(* IEC 61131-3 sources: Industry-PLC-LLM/data/PLCBEAD_repo/PLCBEAD_PLCEmbed-main/PLC-BEAD/Source/OpenPLCv2 (part 3) *)

(* ---- CEXP.ST ---- *)
TYPE oscat_complex :
  STRUCT
	re : REAL;
	im : REAL;
  END_STRUCT;
END_TYPE

FUNCTION_BLOCK CEXP_Block
	VAR_INPUT
		X :	oscat_complex;
	END_VAR

	VAR_OUTPUT
		CEXP :	oscat_complex;
	END_VAR

	VAR
		Temp :	REAL;
	END_VAR

	temp := EXP(X.re);
	CEXP.re := temp * COS(X.im);
	CEXP.im := temp * SIN(X.im);

END_FUNCTION_BLOCK

PROGRAM program0
  VAR
    LocalVar0 : oscat_complex;
	LocalOUT  : oscat_complex;
	func_block : CEXP_Block;
  END_VAR
	func_block.X  := LocalVar0;
	func_block();
	LocalOUT := func_block.CEXP;
END_PROGRAM

CONFIGURATION Config0
  RESOURCE Res0 ON PLC
    TASK task0(INTERVAL := T#20ms,PRIORITY := 0);
    PROGRAM instance0 WITH task0 : program0;
  END_RESOURCE
END_CONFIGURATION

(* ---- CHARNAME.ST ---- *)
TYPE
  oscat_CHARNAMES	: ARRAY [1..11] OF STRING;
END_TYPE

FUNCTION_BLOCK SETUP_CHARNAMES_Block

	VAR_IN_OUT
		CHARNAMES :	oscat_CHARNAMES;
	END_VAR

	VAR
		init :	BOOL;
	END_VAR

	IF init THEN RETURN; END_IF;

	init := TRUE;

	CHARNAMES[01] := '123';
	CHARNAMES[02] := '456';
	CHARNAMES[03] := 'zgsdafasf';
	CHARNAMES[04] := 'sadfsdfa';
	CHARNAMES[05] := 'asdfdsafdfds';
	CHARNAMES[06] := 'sadfsdfsdf';
	CHARNAMES[07] := 'sfsfdfdddd';
	CHARNAMES[08] := 'dddddted';
	CHARNAMES[10] := 'wer';
	CHARNAMES[11] := 'werwer';

END_FUNCTION_BLOCK

FUNCTION_BLOCK CHR_TO_STRING_Block
	VAR_INPUT
		C :	BYTE;
	END_VAR

	VAR_OUTPUT
		CHR_TO_STRING :	STRING;
	END_VAR

	CHR_TO_STRING := BYTE_TO_STRING(C);

END_FUNCTION_BLOCK

FUNCTION_BLOCK CHARNAME_Block

	VAR_INPUT
		C :	BYTE;
	END_VAR

	VAR_OUTPUT
		CHARNAME :	STRING;
	END_VAR

	VAR
		CHARNAME2 :	STRING;
		pos :	INT;
		i :	INT;
		CHR_TO_STRING :	CHR_TO_STRING_Block;
		SETUP_CHARNAMES :	SETUP_CHARNAMES_Block;
		CHARNAMES :	oscat_CHARNAMES;
	END_VAR

	SETUP_CHARNAMES(CHARNAMES:=CHARNAMES);
	CHARNAMES:=SETUP_CHARNAMES.CHARNAMES;

	IF C <> BYTE#0 THEN
		(* construct search string from code followed by $ sign, also clear charname string*)
		CHR_TO_STRING(C:=C);
		CHARNAME := CHR_TO_STRING.CHR_TO_STRING;
		CHARNAME2 := CONCAT(CHARNAME,'&');
		CHARNAME := CONCAT(';', CHARNAME2);
		WHILE pos = 0 AND (i < 11) DO
			i := i + 1;
			pos := FIND(CHARNAMES[i], CHARNAME);
		END_WHILE;
		IF pos > 0 THEN
			CHARNAME := MID(CHARNAMES[i], 10, pos + 3);
			(* search for end of name and truncate *)
			pos := FIND(CHARNAME, ';');
			CHARNAME := LEFT(CHARNAME,pos - 1);
		ELSE
			CHR_TO_STRING(C:=C);
			CHARNAME := CHR_TO_STRING.CHR_TO_STRING;
		END_IF;
	ELSE
		CHARNAME := '';
	END_IF;

END_FUNCTION_BLOCK

PROGRAM program0
  VAR
	C :	BYTE;
	CHARNAME :	STRING;
	func_block : CHARNAME_Block;
  END_VAR
	func_block.C  :=C ;
	func_block();
	CHARNAME := func_block.CHARNAME;
END_PROGRAM

CONFIGURATION Config0
	RESOURCE Res0 ON PLC
		TASK task0(INTERVAL := T#20ms,PRIORITY := 0);
		PROGRAM instance0 WITH task0 : program0;
	END_RESOURCE
END_CONFIGURATION

(* ---- CHR_TO_STRING.ST ---- *)
FUNCTION_BLOCK CHR_TO_STRING_Block
	VAR_INPUT
		C :	BYTE;
	END_VAR

	VAR_OUTPUT
		CHR_TO_STRING :	STRING;
	END_VAR

	CHR_TO_STRING := BYTE_TO_STRING(C);

END_FUNCTION_BLOCK

PROGRAM program0
  VAR
    LocalVar0 : BYTE;
	LocalOUT  : STRING;
	func_block : CHR_TO_STRING_Block;
  END_VAR
	func_block.C  := LocalVar0;
	func_block();
	LocalOUT := func_block.CHR_TO_STRING;
END_PROGRAM

CONFIGURATION Config0
  RESOURCE Res0 ON PLC
    TASK task0(INTERVAL := T#20ms,PRIORITY := 0);
    PROGRAM instance0 WITH task0 : program0;
  END_RESOURCE
END_CONFIGURATION

(* ---- CINV.ST ---- *)
TYPE oscat_complex :
  STRUCT
	re : REAL;
	im : REAL;
  END_STRUCT;
END_TYPE

FUNCTION_BLOCK CINV_Block

	VAR_INPUT
		X :	oscat_complex;
	END_VAR

	VAR_OUTPUT
		CINV :	oscat_complex;
	END_VAR

	VAR
		temp :	REAL;
	END_VAR

	temp := X.re * X.re + X.im * X.im;
	IF temp = 0.0 THEN CINV.re := 0.0;CINV.im := 0.0;RETURN;END_IF;
	CINV.re := X.re / temp;
	CINV.im := -X.im / temp;

END_FUNCTION_BLOCK

PROGRAM program0
  VAR
    LocalVar0 : oscat_complex;
	LocalOUT  : oscat_complex;
	func_block : CINV_Block;
  END_VAR
	func_block.X  := LocalVar0;
	func_block();
	LocalOUT := func_block.CINV;
END_PROGRAM

CONFIGURATION Config0
  RESOURCE Res0 ON PLC
    TASK task0(INTERVAL := T#20ms,PRIORITY := 0);
    PROGRAM instance0 WITH task0 : program0;
  END_RESOURCE
END_CONFIGURATION

(* ---- CLEAN.ST ---- *)
FUNCTION_BLOCK CLEAN_Block
	VAR_INPUT
		IN :	STRING;
		CX :	STRING;
	END_VAR

	VAR_OUTPUT
		CLEAN :	STRING;
	END_VAR

	VAR
		pos :	INT;
		stop :	INT;
		char :	STRING;
	END_VAR

	CLEAN := IN;
	stop := LEN(in);
	pos := 1;
	WHILE pos <= stop DO
		char := MID(CLEAN, 1, pos);
		IF FIND(cx,char) > 0 THEN
			pos := pos + 1;
		ELSE
			CLEAN := DELETE(CLEAN, 1, pos);
			stop := stop - 1;
		END_IF;
	END_WHILE;

END_FUNCTION_BLOCK

PROGRAM program0
  VAR
    LocalVar0 : STRING;
    LocalVar1 : STRING;
	LocalOUT  : STRING;
	func_block : CLEAN_Block;
  END_VAR
	func_block.IN  := LocalVar0;
	func_block.CX := LocalVar1;
	func_block();
	LocalOUT := func_block.CLEAN;

END_PROGRAM

CONFIGURATION Config0
  RESOURCE Res0 ON PLC
    TASK task0(INTERVAL := T#20ms,PRIORITY := 0);
    PROGRAM instance0 WITH task0 : program0;
  END_RESOURCE
END_CONFIGURATION

(* ---- CLICK.ST ---- *)
FUNCTION_BLOCK SW_RECONFIG_Block

	VAR_INPUT
		IN :	BOOL;
		TD :	TIME;
		TR :	TIME;
	END_VAR

	VAR_OUTPUT
		Q :	BOOL;
	END_VAR

	VAR
		T1 :	TON;
		T2 :	TON;
		INV :	BOOL;
	END_VAR

	t1(in := IN, PT := TD);

	IF tr > t#0s THEN
		Q := t1.Q XOR inv;
		T2(in := Q, pt := TR);
		IF T2.Q THEN INV := NOT INV; END_IF;
	ELSE
		Q := t1.Q;
	END_IF;

END_FUNCTION_BLOCK

FUNCTION UDINT_TO_TIME2:TIME

	VAR_INPUT
		IN :	UDINT;
	END_VAR

	UDINT_TO_TIME2 := DINT_TO_TIME(UDINT_TO_DINT(IN));

END_FUNCTION

FUNCTION_BLOCK T_PLC_MS_block
	VAR_OUTPUT
		T_PLC_MS :	UDINT;
	END_VAR

	VAR_EXTERNAL
		PLC_TICKS_PER_SEC :	INT;
		PLC_SYS_TICK_CNT :	DINT;
	END_VAR

	VAR
		debug :	BOOL;(*Debug-Mode ON / OFF*)
		N :	INT;(*Debug-Faktor*)
		Offset :	UDINT;(*Debug-Offset*)
		temp :	DWORD := DWORD#1;(*Debug-Offset*)
		mode :	BOOL;(*modus*)
		faktor :	UDINT;(*Systemtakt-Faktor*)
		init :	BOOL;
		v_plc_ticks_per_sec :	UDINT;
		base :	UDINT := UDINT#1000;
	END_VAR

	IF init = FALSE THEN
		v_plc_ticks_per_sec := INT_TO_UDINT(PLC_TICKS_PER_SEC);
		IF v_plc_ticks_per_sec = UDINT#1024 THEN
			faktor := UDINT#1;
			mode := FALSE;
		ELSIF v_plc_ticks_per_sec > UDINT#0 THEN
			IF v_plc_ticks_per_sec <= base THEN
				faktor := base / v_plc_ticks_per_sec;
				mode := FALSE;
			ELSE
				faktor := v_plc_ticks_per_sec / base;
				mode := TRUE;
			END_IF;
		ELSE
			faktor := UDINT#1;
		END_IF;
		init := TRUE;
	END_IF;

	IF mode THEN
		T_PLC_MS := DINT_TO_UDINT(PLC_SYS_TICK_CNT) / faktor;
	ELSE
		T_PLC_MS := DINT_TO_UDINT(PLC_SYS_TICK_CNT) * faktor;
	END_IF;

	IF debug THEN
		T_PLC_MS := (DWORD_TO_UDINT(SHL(UDINT_TO_DWORD(T_PLC_MS),N) OR SHL(temp,N)) - UDINT#1) + Offset;
	END_IF;

END_FUNCTION_BLOCK

FUNCTION_BLOCK CLICK_Block

	VAR_INPUT
		IN :	BOOL;
		T_DEBOUNCE :	TIME := T#10ms;
		T_SHORT :	TIME := T#200ms;
		T_PAUSE :	TIME := T#500ms;
		T_RECONFIG :	TIME := T#1m;
	END_VAR

	VAR_OUTPUT
		Q :	BOOL;
		SINGLE :	BOOL;
		DOUBLE :	BOOL;
		TRIPLE :	BOOL;
		STATUS :	BYTE;
	END_VAR

	VAR
		s_in :	SW_RECONFIG_Block;
		tx :	TIME;
		state :	INT;
		last :	TIME;
		T_PLC_MS :	T_PLC_MS_Block;
	END_VAR

	s_in(in := in, TD := T_debounce, TR := T_reconfig);

	T_PLC_MS();
	tx:= UDINT_TO_TIME(T_PLC_MS.T_PLC_MS);

	IF s_in.Q XOR Q THEN
		last := tx;
		IF s_in.Q THEN state := state + 1; END_IF;
	END_IF;
	Q := s_in.Q;

	IF state > 0 THEN
		IF (Q AND tx - last > t_short) OR (NOT Q AND tx - last > t_pause) THEN
			CASE state OF
				1:	single := TRUE;
					status := BYTE#111;
				2:	double := TRUE;
					status := BYTE#112;
				3:	triple := TRUE;
					status := BYTE#113;
			END_CASE;
			state := 0;
		END_IF;
	ELSIF NOT q THEN
		single := FALSE;
		double := FALSE;
		triple := FALSE;
		status := BYTE#110;
		last := tx;
		state := 0;
	END_IF;

END_FUNCTION_BLOCK

PROGRAM program0
	VAR
		IN :	BOOL;
		T_DEBOUNCE :	TIME := T#10ms;
		T_SHORT :	TIME := T#200ms;
		T_PAUSE :	TIME := T#500ms;
		T_RECONFIG :	TIME := T#1m;
		Q :	BOOL;
		SINGLE :	BOOL;
		DOUBLE :	BOOL;
		TRIPLE :	BOOL;
		STATUS :	BYTE;

		func_block : CLICK_Block;
	END_VAR
	func_block.IN := IN;
	func_block.T_DEBOUNCE := T_DEBOUNCE;
	func_block.T_SHORT := T_SHORT;
	func_block.T_PAUSE := T_PAUSE;
	func_block.T_RECONFIG := T_RECONFIG;

	func_block();
	Q  := func_block.Q;
	SINGLE  := func_block.SINGLE;
	DOUBLE  := func_block.DOUBLE;
	TRIPLE  := func_block.TRIPLE;
	STATUS  := func_block.STATUS;
END_PROGRAM

CONFIGURATION Config0
	VAR_GLOBAL
		PLC_TICKS_PER_SEC :	INT;
		PLC_SYS_TICK_CNT :	DINT;
	END_VAR
  	RESOURCE Res0 ON PLC
    	TASK task0(INTERVAL := T#20ms,PRIORITY := 0);
    	PROGRAM instance0 WITH task0 : program0;
  	END_RESOURCE
END_CONFIGURATION

(* ---- CLICK_CNT.ST ---- *)
FUNCTION_BLOCK CLICK_CNT
	VAR_INPUT
		IN :	BOOL;
		N :	INT;
		TC :	TIME;
	END_VAR

	VAR_OUTPUT
		Q :	BOOL;
	END_VAR

	VAR
		tx :	TP;
		edge :	BOOL;
		cnt :	INT := INT#-1;
	END_VAR

	Q := FALSE;

	IF in AND NOT edge AND NOT tx.q THEN
		cnt := 0;
	ELSIF tx.Q AND NOT IN AND edge THEN
		cnt := cnt + 1;
	ELSIF NOT tx.Q THEN
		Q := cnt=N;
		cnt := -1;
	END_IF;
	edge := IN;
	tx(in := IN, pt := TC);
END_FUNCTION_BLOCK

PROGRAM program0
  VAR
    LocalVar0 : BOOl;
    LocalVar1 : INT;
	LocalVar2 : TIME;
	LocalOUT  : BOOL;
	func_block : CLICK_CNT;
  END_VAR
	func_block.IN  := LocalVar0;
	func_block.N := LocalVar1;
	func_block.TC  := LocalVar2;
	func_block();
	LocalOUT := func_block.Q;

END_PROGRAM

CONFIGURATION Config0
  RESOURCE Res0 ON PLC
    TASK task0(INTERVAL := T#20ms,PRIORITY := 0);
    PROGRAM instance0 WITH task0 : program0;
  END_RESOURCE
END_CONFIGURATION

(* ---- CLICK_DEC.ST ---- *)
FUNCTION_BLOCK CLICK_DEC

	VAR_INPUT
		IN :	BOOL;
		TC :	TIME;
	END_VAR

	VAR_OUTPUT
		Q0 :	BOOL;
		Q1 :	BOOL;
		Q2 :	BOOL;
		Q3 :	BOOL;
	END_VAR

	VAR
		tx :	TP;
		edge :	BOOL;
		cnt :	INT := INT#-1;
	END_VAR

	IF in = FALSE THEN
		Q0 := FALSE;
		Q1 := FALSE;
		Q2 := FALSE;
		Q3 := FALSE;
	END_IF;

	IF in AND NOT edge AND NOT tx.q THEN
		cnt := 0;
	ELSIF tx.Q AND NOT IN AND edge THEN
		cnt := cnt + 1;
	ELSIF NOT tx.Q THEN
		CASE cnt OF
			0 : Q0 := TRUE;
			1 : Q1 := TRUE;
			2 : Q2 := TRUE;
			3 : Q3 := TRUE;
		END_CASE;
		cnt := -1;
	END_IF;

	edge := IN;
	tx(in := IN, pt := TC);

END_FUNCTION_BLOCK

PROGRAM program0
  VAR
    LocalVar0 : BOOL;
    LocalVar1 : TIME;
	Q0 :	BOOL;
	Q1 :	BOOL;
	Q2 :	BOOL;
	Q3 :	BOOL;
	func_block : CLICK_DEC;
  END_VAR
	func_block.IN  := LocalVar0;
	func_block.TC := LocalVar1;
	func_block();
	Q0 := func_block.Q0;
	Q1 := func_block.Q1;
	Q2 := func_block.Q2;
	Q3 := func_block.Q3;
END_PROGRAM

CONFIGURATION Config0
  RESOURCE Res0 ON PLC
    TASK task0(INTERVAL := T#20ms,PRIORITY := 0);
    PROGRAM instance0 WITH task0 : program0;
  END_RESOURCE
END_CONFIGURATION

(* ---- CLICK_MODE.ST ---- *)
FUNCTION_BLOCK CLICK_MODE_Block

	VAR_INPUT
		IN :	BOOL;
		T_LONG :	TIME := T#500ms;
	END_VAR

	VAR_OUTPUT
		SINGLE :	BOOL;
		DOUBLE :	BOOL;
		LONG :	BOOL;
		TP_LONG :	BOOL;
	END_VAR

	VAR
		Timer :	TP;
		cnt :	INT;
		last :	BOOL;
	END_VAR

	timer(in := IN, PT := T_LONG);
	single := FALSE;
	double := FALSE;

	IF timer.Q THEN
		IF NOT in AND last THEN	cnt := cnt + 1; END_IF;
	ELSE
		CASE cnt OF
			1 : single := TRUE;
			2 : double := TRUE;
		END_CASE;
		cnt := 0;
	END_IF;
	last := in;
	TP_LONG := NOT timer.Q AND (NOT LONG) AND IN;
	LONG := NOT timer.Q AND in;

END_FUNCTION_BLOCK

PROGRAM program0
	VAR
		IN :	BOOL;
		T_LONG :	TIME := T#500ms;
		SINGLE :	BOOL;
		DOUBLE :	BOOL;
		LONG :	BOOL;
		TP_LONG :	BOOL;

		func_block : CLICK_MODE_Block;
	END_VAR
	func_block.IN := IN;
	func_block.T_LONG := T_LONG;

	func_block();
	SINGLE  := func_block.SINGLE;
	DOUBLE  := func_block.DOUBLE;
	LONG  := func_block.LONG;
	TP_LONG  := func_block.TP_LONG;
END_PROGRAM

CONFIGURATION Config0
	RESOURCE Res0 ON PLC
		TASK task0(INTERVAL := T#20ms,PRIORITY := 0);
		PROGRAM instance0 WITH task0 : program0;
	END_RESOURCE
END_CONFIGURATION

(* ---- CLK_DIV.ST ---- *)
FUNCTION BIT_OF_DWORD : BOOL
  VAR_INPUT
    IN : DWORD;
    N : INT;
  END_VAR

  BIT_OF_DWORD := (SHR(in,N) AND 16#00000001) > 0;
  (* from OSCAT library; www.oscat.de  *)
END_FUNCTION

FUNCTION_BLOCK CLK_DIV
	VAR_INPUT
		CLK :	BOOL;
		RST :	BOOL;
	END_VAR

	VAR_OUTPUT
		Q0 :	BOOL := FALSE;
		Q1 :	BOOL := FALSE;
		Q2 :	BOOL := FALSE;
		Q3 :	BOOL := FALSE;
		Q4 :	BOOL := FALSE;
		Q5 :	BOOL := FALSE;
		Q6 :	BOOL := FALSE;
		Q7 :	BOOL := FALSE;
	END_VAR

	VAR
		cnt :	BYTE := 0;
	END_VAR

	IF rst THEN
		cnt:= BYTE#0;
		Q0 := FALSE;
		Q1 := FALSE;
		Q2 := FALSE;
		Q3 := FALSE;
		Q4 := FALSE;
		Q5 := FALSE;
		Q6 := FALSE;
		Q7 := FALSE;
	ELSIF clk THEN
		cnt:= USINT_TO_BYTE(BYTE_TO_USINT(cnt) + USINT#1);

		Q0 := BIT_OF_DWORD(BYTE_TO_DWORD(cnt),0); (* Q0 := cnt.X0; *)
		Q1 := BIT_OF_DWORD(BYTE_TO_DWORD(cnt),1); (* Q1 := cnt.X1; *)
		Q2 := BIT_OF_DWORD(BYTE_TO_DWORD(cnt),2); (* Q2 := cnt.X2; *)
		Q3 := BIT_OF_DWORD(BYTE_TO_DWORD(cnt),3); (* Q3 := cnt.X3; *)
		Q4 := BIT_OF_DWORD(BYTE_TO_DWORD(cnt),4); (* Q4 := cnt.X4; *)
		Q5 := BIT_OF_DWORD(BYTE_TO_DWORD(cnt),5); (* Q5 := cnt.X5; *)
		Q6 := BIT_OF_DWORD(BYTE_TO_DWORD(cnt),6); (* Q6 := cnt.X6; *)
		Q7 := BIT_OF_DWORD(BYTE_TO_DWORD(cnt),7); (* Q7 := cnt.X7; *)

	END_IF;

END_FUNCTION_BLOCK

PROGRAM program0
  VAR
    LocalVar0 : BOOL;
    LocalVar1 : BOOL;
	Q0 :	BOOL;
	Q1 :	BOOL;
	Q2 :	BOOL;
	Q3 :	BOOL;
	Q4 :	BOOL;
	Q5 :	BOOL;
	Q6 :	BOOL;
	Q7 :	BOOL;
	func_block : CLK_DIV;
  END_VAR
	func_block.CLK  := LocalVar0;
	func_block.RST := LocalVar1;
	func_block();
	Q0 := func_block.Q0;
	Q1 := func_block.Q1;
	Q2 := func_block.Q2;
	Q3 := func_block.Q3;
	Q4 := func_block.Q4;
	Q5 := func_block.Q5;
	Q6 := func_block.Q6;
	Q7 := func_block.Q7;
END_PROGRAM

CONFIGURATION Config0
  RESOURCE Res0 ON PLC
    TASK task0(INTERVAL := T#20ms,PRIORITY := 0);
    PROGRAM instance0 WITH task0 : program0;
  END_RESOURCE
END_CONFIGURATION

(* ---- CLK_N.ST ---- *)
FUNCTION_BLOCK T_PLC_MS_block
	VAR_OUTPUT
		T_PLC_MS :	UDINT;
	END_VAR

	VAR_EXTERNAL
		PLC_TICKS_PER_SEC :	INT;
		PLC_SYS_TICK_CNT :	DINT;
	END_VAR

	VAR
		debug :	BOOL;(*Debug-Mode ON / OFF*)
		N :	INT;(*Debug-Faktor*)
		Offset :	UDINT;(*Debug-Offset*)
		temp :	DWORD := DWORD#1;(*Debug-Offset*)
		mode :	BOOL;(*modus*)
		faktor :	UDINT;(*Systemtakt-Faktor*)
		init :	BOOL;
		v_plc_ticks_per_sec :	UDINT;
		base :	UDINT := UDINT#1000;
	END_VAR

	IF init = FALSE THEN
		v_plc_ticks_per_sec := INT_TO_UDINT(PLC_TICKS_PER_SEC);
		IF v_plc_ticks_per_sec = UDINT#1024 THEN
			faktor := UDINT#1;
			mode := FALSE;
		ELSIF v_plc_ticks_per_sec > UDINT#0 THEN
			IF v_plc_ticks_per_sec <= base THEN
				faktor := base / v_plc_ticks_per_sec;
				mode := FALSE;
			ELSE
				faktor := v_plc_ticks_per_sec / base;
				mode := TRUE;
			END_IF;
		ELSE
			faktor := UDINT#1;
		END_IF;
		init := TRUE;
	END_IF;

	IF mode THEN
		T_PLC_MS := DINT_TO_UDINT(PLC_SYS_TICK_CNT) / faktor;
	ELSE
		T_PLC_MS := DINT_TO_UDINT(PLC_SYS_TICK_CNT) * faktor;
	END_IF;

	IF debug THEN
		T_PLC_MS := (DWORD_TO_UDINT(SHL(UDINT_TO_DWORD(T_PLC_MS),N) OR SHL(temp,N)) - UDINT#1) + Offset;
	END_IF;

END_FUNCTION_BLOCK

FUNCTION BIT_OF_DWORD:BOOL
	VAR_INPUT
		IN :	DWORD;
		N :	INT;
	END_VAR
	BIT_OF_DWORD := (SHR(in,n) AND DWORD#1) > DWORD#0;
END_FUNCTION

FUNCTION_BLOCK CLK_N
	VAR_INPUT
		N :	INT;
	END_VAR

	VAR_OUTPUT
		Q :	BOOL;
	END_VAR

	VAR
		T_PLC_MS :	T_PLC_MS_block;
		edge :	BOOL;
		clk :	BOOL;
	END_VAR

	T_PLC_MS();
	clk := BIT_OF_DWORD(SHR(UDINT_TO_DWORD(T_PLC_MS.T_PLC_MS),N),0);
	Q := clk XOR edge;
	edge := clk;
END_FUNCTION_BLOCK

PROGRAM program0
  VAR
    LocalVar0 : INT;
	LocalOUT  : BOOL;
	func_block : CLK_N;
  END_VAR
	func_block.N  := LocalVar0;
	func_block();
	LocalOUT := func_block.Q;

END_PROGRAM

CONFIGURATION Config0
	VAR_GLOBAL
		PLC_TICKS_PER_SEC :	INT;
		PLC_SYS_TICK_CNT :	DINT;
	END_VAR

  RESOURCE Res0 ON PLC
    TASK task0(INTERVAL := T#20ms,PRIORITY := 0);
    PROGRAM instance0 WITH task0 : program0;
  END_RESOURCE
END_CONFIGURATION

(* ---- CLK_PRG.ST ---- *)
FUNCTION_BLOCK T_PLC_MS_block
	VAR_OUTPUT
		T_PLC_MS :	UDINT;
	END_VAR

	VAR_EXTERNAL
		PLC_TICKS_PER_SEC :	INT;
		PLC_SYS_TICK_CNT :	DINT;
	END_VAR

	VAR
		debug :	BOOL;(*Debug-Mode ON / OFF*)
		N :	INT;(*Debug-Faktor*)
		Offset :	UDINT;(*Debug-Offset*)
		temp :	DWORD := DWORD#1;(*Debug-Offset*)
		mode :	BOOL;(*modus*)
		faktor :	UDINT;(*Systemtakt-Faktor*)
		init :	BOOL;
		v_plc_ticks_per_sec :	UDINT;
		base :	UDINT := UDINT#1000;
	END_VAR

	IF init = FALSE THEN
		v_plc_ticks_per_sec := INT_TO_UDINT(PLC_TICKS_PER_SEC);
		IF v_plc_ticks_per_sec = UDINT#1024 THEN
			faktor := UDINT#1;
			mode := FALSE;
		ELSIF v_plc_ticks_per_sec > UDINT#0 THEN
			IF v_plc_ticks_per_sec <= base THEN
				faktor := base / v_plc_ticks_per_sec;
				mode := FALSE;
			ELSE
				faktor := v_plc_ticks_per_sec / base;
				mode := TRUE;
			END_IF;
		ELSE
			faktor := UDINT#1;
		END_IF;
		init := TRUE;
	END_IF;

	IF mode THEN
		T_PLC_MS := DINT_TO_UDINT(PLC_SYS_TICK_CNT) / faktor;
	ELSE
		T_PLC_MS := DINT_TO_UDINT(PLC_SYS_TICK_CNT) * faktor;
	END_IF;

	IF debug THEN
		T_PLC_MS := (DWORD_TO_UDINT(SHL(UDINT_TO_DWORD(T_PLC_MS),N) OR SHL(temp,N)) - UDINT#1) + Offset;
	END_IF;

END_FUNCTION_BLOCK

FUNCTION_BLOCK CLK_PRG
	VAR_INPUT
		PT :	TIME := T#10ms;
	END_VAR

	VAR_OUTPUT
		Q :	BOOL;
	END_VAR

	VAR
		init :	BOOL := FALSE;
		last :	TIME;
		tx :	TIME;
		T_PLC_MS :	T_PLC_MS_block;
	END_VAR

	T_PLC_MS();
	tx:= UDINT_TO_TIME(T_PLC_MS.T_PLC_MS);

	IF NOT init THEN
		init := TRUE;
		last := tx - pt;
	END_IF;

	Q := tx - last >= pt;
	IF Q THEN last := tx; END_IF;
END_FUNCTION_BLOCK

PROGRAM program0
  VAR
    LocalVar0 : TIME;
	LocalOUT  : BOOL;
	func_block : CLK_PRG;
  END_VAR
	func_block.PT  := LocalVar0;
	func_block();
	LocalOUT := func_block.Q;

END_PROGRAM

CONFIGURATION Config0
	VAR_GLOBAL
		PLC_TICKS_PER_SEC :	INT;
		PLC_SYS_TICK_CNT :	DINT;
	END_VAR

  RESOURCE Res0 ON PLC
    TASK task0(INTERVAL := T#20ms,PRIORITY := 0);
    PROGRAM instance0 WITH task0 : program0;
  END_RESOURCE
END_CONFIGURATION

(* ---- CLK_PULSE.ST ---- *)
FUNCTION_BLOCK T_PLC_MS_block
	VAR_OUTPUT
		T_PLC_MS :	UDINT;
	END_VAR

	VAR_EXTERNAL
		PLC_TICKS_PER_SEC :	INT;
		PLC_SYS_TICK_CNT :	DINT;
	END_VAR

	VAR
		debug :	BOOL;(*Debug-Mode ON / OFF*)
		N :	INT;(*Debug-Faktor*)
		Offset :	UDINT;(*Debug-Offset*)
		temp :	DWORD := DWORD#1;(*Debug-Offset*)
		mode :	BOOL;(*modus*)
		faktor :	UDINT;(*Systemtakt-Faktor*)
		init :	BOOL;
		v_plc_ticks_per_sec :	UDINT;
		base :	UDINT := UDINT#1000;
	END_VAR

	IF init = FALSE THEN
		v_plc_ticks_per_sec := INT_TO_UDINT(PLC_TICKS_PER_SEC);
		IF v_plc_ticks_per_sec = UDINT#1024 THEN
			faktor := UDINT#1;
			mode := FALSE;
		ELSIF v_plc_ticks_per_sec > UDINT#0 THEN
			IF v_plc_ticks_per_sec <= base THEN
				faktor := base / v_plc_ticks_per_sec;
				mode := FALSE;
			ELSE
				faktor := v_plc_ticks_per_sec / base;
				mode := TRUE;
			END_IF;
		ELSE
			faktor := UDINT#1;
		END_IF;
		init := TRUE;
	END_IF;

	IF mode THEN
		T_PLC_MS := DINT_TO_UDINT(PLC_SYS_TICK_CNT) / faktor;
	ELSE
		T_PLC_MS := DINT_TO_UDINT(PLC_SYS_TICK_CNT) * faktor;
	END_IF;

	IF debug THEN
		T_PLC_MS := (DWORD_TO_UDINT(SHL(UDINT_TO_DWORD(T_PLC_MS),N) OR SHL(temp,N)) - UDINT#1) + Offset;
	END_IF;

END_FUNCTION_BLOCK

FUNCTION TIME_TO_UDINT2:UDINT
	VAR_INPUT
		X :	TIME;
	END_VAR

	TIME_TO_UDINT2 := DINT_TO_UDINT(TIME_TO_DINT(X));
END_FUNCTION

FUNCTION_BLOCK CLK_PULSE
	VAR_INPUT
		PT :	TIME;
		N :	INT;
		RST :	BOOL;
	END_VAR

	VAR_OUTPUT
		Q :	BOOL;
		CNT :	INT;
		RUN :	BOOL;
	END_VAR

	VAR
		tx :	UDINT;
		tn :	UDINT;
		init :	BOOL;
		T_PLC_MS :	T_PLC_MS_block;
	END_VAR

	T_PLC_MS();
	tx:= T_PLC_MS.T_PLC_MS;
	Q := FALSE;				(* reset Q we generate pulses only for one cycle *)
	RUN := CNT < N;

	IF NOT init OR RST THEN
		init := TRUE;
		CNT := 0;
		tn := tx - TIME_TO_UDINT2(PT);
		RUN := FALSE;
	ELSIF (cnt < N OR N = 0) AND tx - tn >= TIME_TO_UDINT2(PT) THEN		(* generate a pulse *)
		CNT := CNT + 1;
		Q := TRUE;
		tn := tn + TIME_TO_UDINT2(PT);
	END_IF;

END_FUNCTION_BLOCK

PROGRAM program0
  VAR
    LocalVar0 : TIME;
	LocalVar1 : INT;
	LocalVar2 : BOOL;

	Q :	BOOL;
	CNT :	INT;
	RUN :	BOOL;
	func_block : CLK_PULSE;
  END_VAR
	func_block.PT  := LocalVar0;
	func_block.N  := LocalVar1;
	func_block.RST  := LocalVar2;
	func_block();
	Q:= func_block.Q;
	CNT := func_block.CNT;
	RUN := func_block.RUN;

END_PROGRAM

CONFIGURATION Config0
	VAR_GLOBAL
		PLC_TICKS_PER_SEC :	INT;
		PLC_SYS_TICK_CNT :	DINT;
	END_VAR

  RESOURCE Res0 ON PLC
    TASK task0(INTERVAL := T#20ms,PRIORITY := 0);
    PROGRAM instance0 WITH task0 : program0;
  END_RESOURCE
END_CONFIGURATION

(* ---- CLOG.ST ---- *)
TYPE oscat_complex :
  STRUCT
	re : REAL;
	im : REAL;
  END_STRUCT;
END_TYPE

FUNCTION ATAN2:REAL
	VAR_INPUT
		X :	REAL;
		Y :	REAL;
	END_VAR

	IF X > 0.0 THEN
		ATAN2 := ATAN(Y/X);
	ELSIF X < 0.0 THEN
		IF Y >= 0.0 THEN
			ATAN2 := ATAN(Y/X) + 3.14159265358979323846264338327950288;
		ELSE
			ATAN2 := ATAN(Y/X) - 3.14159265358979323846264338327950288;
		END_IF;
	ELSIF Y > 0.0 THEN
		ATAN2 := 1.5707963267948965580;
	ELSIF Y < 0.0 THEN
		ATAN2 := -1.5707963267948965580;
	ELSE
		ATAN2 := 0.0;
	END_IF;

END_FUNCTION

FUNCTION HYPOT:REAL
	VAR_INPUT
		X :	REAL;
		Y :	REAL;
	END_VAR

	HYPOT := SQRT(x*x + y*y);
END_FUNCTION

FUNCTION_BLOCK CLOG_Block

	VAR_INPUT
		X :	oscat_complex;
	END_VAR

	VAR_OUTPUT
		CLOG :	oscat_complex;
	END_VAR

	CLOG.re := LN(HYPOT(X.re, X.im));
	CLOG.im := ATAN2(X.im, X.re);

END_FUNCTION_BLOCK

PROGRAM program0
  VAR
    LocalVar0 : oscat_complex;
	LocalOUT  : oscat_complex;
	func_block : CLOG_Block;
  END_VAR
	func_block.X  := LocalVar0;
	func_block();
	LocalOUT := func_block.CLOG;
END_PROGRAM

CONFIGURATION Config0
  RESOURCE Res0 ON PLC
    TASK task0(INTERVAL := T#20ms,PRIORITY := 0);
    PROGRAM instance0 WITH task0 : program0;
  END_RESOURCE
END_CONFIGURATION

(* ---- CMUL.ST ---- *)
TYPE oscat_complex :
  STRUCT
	re : REAL;
	im : REAL;
  END_STRUCT;
END_TYPE

FUNCTION_BLOCK CMUL_Block

	VAR_INPUT
		X :	oscat_complex;
		Y :	oscat_complex;
	END_VAR

	VAR_OUTPUT
		CMUL :	oscat_complex;
	END_VAR

	CMUL.re := X.re * Y.re - X.im * Y.im;
	CMUL.im := X.re * Y.im + X.im * Y.re;
END_FUNCTION_BLOCK

PROGRAM program0
  VAR
    LocalVar0 : oscat_complex;
	LocalVar1 : oscat_complex;
	LocalOUT  : oscat_complex;
	func_block : CMUL_Block;
  END_VAR
	func_block.X  := LocalVar0;
	func_block.Y  := LocalVar1;
	func_block();
	LocalOUT := func_block.CMUL;
END_PROGRAM

CONFIGURATION Config0
  RESOURCE Res0 ON PLC
    TASK task0(INTERVAL := T#20ms,PRIORITY := 0);
    PROGRAM instance0 WITH task0 : program0;
  END_RESOURCE
END_CONFIGURATION

(* ---- CONTROL_SET1.ST ---- *)
FUNCTION_BLOCK CONTROL_SET1_Block
	VAR_INPUT
		KT :	REAL;
		TT :	REAL;
		PI :	BOOL;
		PIDD :	BOOL;
		P_K :	REAL := 0.5;
		PI_K :	REAL := 0.45;
		PI_TN :	REAL := 0.83;
		PIDD_K :	REAL := 0.6;
		PIDD_TN :	REAL := 0.5;
		PIDD_TV :	REAL := 0.125;
	END_VAR

	VAR_OUTPUT
		KP :	REAL;
		TN :	REAL;
		TV :	REAL;
		KI :	REAL;
		KD :	REAL;
	END_VAR

	IF pi AND PIDD THEN
		KP := 0.0;
		TN := 0.0;
		TV := 0.0;
	ELSIF PIDD THEN
		KP := PIDD_K * Kt;
		TN := PIDD_TN * Tt;
		TV := PIDD_TV * Tt;
	ELSIF PI THEN
		KP := PI_K * Kt;
		TN := PI_TN * Tt;
	ELSE
		KP := P_K * Kt;
	END_IF;
	IF tn > 0.0 THEN KI := KP / TN; ELSE KI := 0.0; END_IF;
	KD := KP * TV;
END_FUNCTION_BLOCK

PROGRAM program0
  VAR
	KT :REAL;
	TT :REAL;
	PI :BOOL;
	PIDD :BOOL;
	P_K :REAL ;
	PI_K :REAL ;
	PI_TN :REAL ;
	PIDD_K :REAL ;
	PIDD_TN :REAL ;
	PIDD_TV :REAL ;
	KP :REAL;
	TN :REAL;
	TV :REAL;
	KI :REAL;
	KD :REAL;
	func_block : CONTROL_SET1_Block;
  END_VAR
	func_block.KT   :=KT  ;
	func_block.TT   :=TT  ;
	func_block.PI   :=PI  ;
	func_block.PIDD   :=PIDD  ;
	func_block.P_K   :=P_K  ;
	func_block.PI_K   :=PI_K  ;
	func_block.PI_TN   :=PI_TN  ;
	func_block.PIDD_K   :=PIDD_K  ;
	func_block.PIDD_TN   :=PIDD_TN  ;
	func_block.PIDD_TV   :=PIDD_TV  ;
	func_block();
	KP := func_block.KP ;
	TN := func_block.TN ;
	TV := func_block.TV ;
	KI := func_block.KI ;
	KD := func_block.KD ;
END_PROGRAM

CONFIGURATION Config0
  RESOURCE Res0 ON PLC
    TASK task0(INTERVAL := T#20ms,PRIORITY := 0);
    PROGRAM instance0 WITH task0 : program0;
  END_RESOURCE
END_CONFIGURATION

(* ---- CONTROL_SET2.ST ---- *)
FUNCTION_BLOCK CONTROL_SET2
	VAR_INPUT
		KS :	REAL;
		TU :	REAL;
		TG :	REAL;
		PI :	BOOL;
		PIDD :	BOOL;
		P_K :	REAL := 1.0;
		PI_K :	REAL := 0.9;
		PI_TN :	REAL := 3.33;
		PIDD_K :	REAL := 1.2;
		PIDD_TN :	REAL := 2.0;
		PIDD_TV :	REAL := 0.5;
	END_VAR

	VAR_OUTPUT
		KP :	REAL;
		TN :	REAL;
		TV :	REAL;
		KI :	REAL;
		KD :	REAL;
	END_VAR

	VAR
		TX :	REAL;
	END_VAR

	IF TU > 0.0 AND KS > 0.0 THEN TX := TG / TU / KS; END_IF;
	IF pi AND PIDD THEN
		KP := 0.0;
		TN := 0.0;
		TV := 0.0;
	ELSIF PIDD THEN
		KP := PIDD_K * TX;
		TN := PIDD_TN * TU;
		TV := PIDD_TV * TU;
	ELSIF PI THEN
		KP := PI_K * TX;
		TN := PI_TN * TU;
	ELSE
		KP := P_K * TX;
	END_IF;

	IF TN > 0.0 THEN KI := KP / TN; ELSE KI := 0.0; END_IF;
	KD := KP * TV;

END_FUNCTION_BLOCK

PROGRAM program0
  VAR
	KS :REAL;
	TG :REAL;
	PI :BOOL;
	PIDD :BOOL;
	P_K :REAL ;
	PI_K :REAL ;
	PI_TN :REAL ;
	PIDD_K :REAL ;
	PIDD_TN :REAL ;
	PIDD_TV :REAL ;
	KP :REAL;
	TN :REAL;
	TV :REAL;
	KI :REAL;
	KD :REAL;
	func_block : CONTROL_SET2;
  END_VAR
	func_block.KS   := KS  ;
	func_block.TG   :=TG  ;
	func_block.PI   :=PI  ;
	func_block.PIDD   :=PIDD  ;
	func_block.P_K   :=P_K  ;
	func_block.PI_K   :=PI_K  ;
	func_block.PI_TN   :=PI_TN  ;
	func_block.PIDD_K   :=PIDD_K  ;
	func_block.PIDD_TN   :=PIDD_TN  ;
	func_block.PIDD_TV   :=PIDD_TV  ;
	func_block();
	KP := func_block.KP ;
	TN := func_block.TN ;
	TV := func_block.TV ;
	KI := func_block.KI ;
	KD := func_block.KD ;
END_PROGRAM

CONFIGURATION Config0
  RESOURCE Res0 ON PLC
    TASK task0(INTERVAL := T#20ms,PRIORITY := 0);
    PROGRAM instance0 WITH task0 : program0;
  END_RESOURCE
END_CONFIGURATION

(* ---- COUNT_BR.ST ---- *)
FUNCTION _BYTE_TO_INT:INT
	VAR_INPUT
		IN :	BYTE;
	END_VAR

	_BYTE_TO_INT := USINT_TO_INT(BYTE_TO_USINT(IN));

END_FUNCTION

FUNCTION INC:INT
	VAR_INPUT
		X :	INT;
		D :	INT;
		M :	INT;
	END_VAR

	inc := (X + D + M + 1) MOD (M + 1);
END_FUNCTION

FUNCTION_BLOCK COUNT_BR
	VAR_INPUT
		SET :	BOOL;
		IN :	BYTE;
		UP :	BOOL;
		DN :	BOOL;
		STEPP :	BYTE := BYTE#1;
		MX :	BYTE := BYTE#255;
		RST :	BOOL;
	END_VAR
	VAR_OUTPUT
		CNT :	BYTE;
	END_VAR

	VAR
		last_up :	BOOL;
		last_dn :	BOOL;
	END_VAR

	IF rst THEN
		cnt := BYTE#0;
	ELSIF set THEN
		cnt := INT_TO_BYTE(LIMIT(0,_BYTE_TO_INT(in),_BYTE_TO_INT(mx)));
	ELSIF up AND NOT last_up THEN
		cnt := INT_TO_BYTE(inc(_BYTE_TO_INT(cnt),_BYTE_TO_INT(stepP),_BYTE_TO_INT(mx)));
	ELSIF dn AND NOT last_dn THEN
		cnt := INT_TO_BYTE(inc(_BYTE_TO_INT(cnt),_BYTE_TO_INT(stepP) * -1,_BYTE_TO_INT(mx)));
	END_IF;
	last_up := up;
	last_dn := dn;
END_FUNCTION_BLOCK

PROGRAM program0
  VAR
	SET :	BOOL;
	IN :	BYTE;
	UP :	BOOL;
	DN :	BOOL;
	STEPP:	BYTE;
	MX :	BYTE;
	RST :	BOOL;

	CNT :	BYTE;
	func_block : COUNT_BR;
  END_VAR
	func_block.SET  :=SET  ;
	func_block.IN   :=IN   ;
	func_block.UP   :=UP   ;
	func_block.DN   :=DN   ;
	func_block.STEPP :=STEPP ;
	func_block.MX   :=MX   ;
	func_block.RST  :=RST  ;

	func_block();
	CNT := func_block.CNT;
END_PROGRAM

CONFIGURATION Config0
  RESOURCE Res0 ON PLC
    TASK task0(INTERVAL := T#20ms,PRIORITY := 0);
    PROGRAM instance0 WITH task0 : program0;
  END_RESOURCE
END_CONFIGURATION

(* ---- COUNT_DR.ST ---- *)
FUNCTION_BLOCK COUNT_DR
	VAR_INPUT
		SET :	BOOL;
		IN :	DWORD;
		UP :	BOOL;
		DN :	BOOL;
		STEPP :	DWORD := DWORD#1;
		MX :	DWORD := DWORD#16#FFFF_FFFF;
		RST :	BOOL;
	END_VAR

	VAR_OUTPUT
		CNT :	DWORD;
	END_VAR

	VAR
		CNT2 :	UDINT;
		STEPP2 :	UDINT;
		MX2 :	UDINT;
		last_up :	BOOL;
		last_dn :	BOOL;
	END_VAR

	STEPP2 := DWORD_TO_UDINT(STEPP);
	MX2   := DWORD_TO_UDINT(MX);
	CNT2  := DWORD_TO_UDINT(CNT);

	IF rst THEN
		CNT2 := UDINT#0;
	ELSIF set THEN
		CNT2 := LIMIT(UDINT#0,DWORD_TO_UDINT(in),mx2);
	ELSIF up AND NOT last_up THEN
		IF STEPP2 > MX2 - CNT2 THEN
			CNT2 := CNT2 - MX2 + STEPP2 - UDINT#1;
		ELSE
			CNT2 := CNT2 + STEPP2;
		END_IF;
	ELSIF dn AND NOT last_dn THEN
		IF STEPP2 > CNT2 THEN
			CNT2 := CNT2 - STEPP2 + MX2 + UDINT#1;
		ELSE
			CNT2 := CNT2 - STEPP2;
		END_IF;
	END_IF;
	last_up := up;
	last_dn := dn;
	CNT := UDINT_TO_DWORD(CNT2);
END_FUNCTION_BLOCK

PROGRAM program0
  VAR
	SET :	BOOL;
	IN :	DWORD;
	UP :	BOOL;
	DN :	BOOL;
	STEPP :	DWORD;
	MX :	DWORD;
	RST :	BOOL;

	CNT :	DWORD;
	func_block : COUNT_DR;
  END_VAR
	func_block.SET  :=SET  ;
	func_block.IN   :=IN   ;
	func_block.UP   :=UP   ;
	func_block.DN   :=DN   ;
	func_block.STEPP :=STEPP ;
	func_block.MX   :=MX   ;
	func_block.RST  :=RST  ;

	func_block();
	CNT := func_block.CNT;
END_PROGRAM

CONFIGURATION Config0
  RESOURCE Res0 ON PLC
    TASK task0(INTERVAL := T#20ms,PRIORITY := 0);
    PROGRAM instance0 WITH task0 : program0;
  END_RESOURCE
END_CONFIGURATION

(* ---- COUNT_SUBSTRING.ST ---- *)
FUNCTION_BLOCK COUNT_SUBSTRING_Block
	VAR_INPUT
		SEARCH :	STRING;
		STR :	STRING;
	END_VAR

	VAR_OUTPUT
		COUNT_SUBSTRING :	INT;
	END_VAR

	VAR
		pos :	INT;
		size :	INT;
	END_VAR

	COUNT_SUBSTRING := 0;
	size := LEN(SEARCH);
	REPEAT
	pos := FIND(STR,SEARCH);
	IF pos > 0 THEN
		STR := REPLACE(STR, '', size,pos);
		COUNT_SUBSTRING := COUNT_SUBSTRING + 1;
	END_IF;
	UNTIL pos = 0
	END_REPEAT;
END_FUNCTION_BLOCK

PROGRAM program0
  VAR
	SEARCH :	STRING;
	STR :	STRING;

	COUNT_SUBSTRING :	INT;
	func_block : COUNT_SUBSTRING_Block;
  END_VAR
	func_block.SEARCH  :=SEARCH  ;
	func_block.STR   :=STR   ;

	func_block();
	COUNT_SUBSTRING := func_block.COUNT_SUBSTRING;
END_PROGRAM

CONFIGURATION Config0
  RESOURCE Res0 ON PLC
    TASK task0(INTERVAL := T#20ms,PRIORITY := 0);
    PROGRAM instance0 WITH task0 : program0;
  END_RESOURCE
END_CONFIGURATION

(* ---- CPOL.ST ---- *)
TYPE oscat_complex :
  STRUCT
	re : REAL;
	im : REAL;
  END_STRUCT;
END_TYPE

FUNCTION_BLOCK CPOL_Block
	VAR_INPUT
		L :	REAL;
		A :	REAL;
	END_VAR

	VAR_OUTPUT
		CPOL :	oscat_complex;
	END_VAR

	CPOL.re := L * COS(A);
	CPOL.im := L * SIN(A);
END_FUNCTION_BLOCK

PROGRAM program0
  VAR
    LocalVar0 : REAL;
	LocalVar1 : REAL;
	CPOL  : oscat_complex;
	func_block : CPOL_Block;
  END_VAR
	func_block.L  := LocalVar0;
	func_block.A  := LocalVar1;
	func_block();
	CPOL := func_block.CPOL;
END_PROGRAM

CONFIGURATION Config0
  RESOURCE Res0 ON PLC
    TASK task0(INTERVAL := T#20ms,PRIORITY := 0);
    PROGRAM instance0 WITH task0 : program0;
  END_RESOURCE
END_CONFIGURATION

(* ---- CPOW.ST ---- *)
TYPE oscat_complex :
  STRUCT
	re : REAL;
	im : REAL;
  END_STRUCT;
END_TYPE

FUNCTION_BLOCK CMUL_Block

	VAR_INPUT
		X :	oscat_complex;
		Y :	oscat_complex;
	END_VAR

	VAR_OUTPUT
		CMUL :	oscat_complex;
	END_VAR

	CMUL.re := X.re * Y.re - X.im * Y.im;
	CMUL.im := X.re * Y.im + X.im * Y.re;
END_FUNCTION_BLOCK

FUNCTION_BLOCK CEXP_Block
	VAR_INPUT
		X :	oscat_complex;
	END_VAR

	VAR_OUTPUT
		CEXP :	oscat_complex;
	END_VAR

	VAR
		Temp :	REAL;
	END_VAR

	temp := EXP(X.re);
	CEXP.re := temp * COS(X.im);
	CEXP.im := temp * SIN(X.im);

END_FUNCTION_BLOCK

FUNCTION ATAN2:REAL
	VAR_INPUT
		X :	REAL;
		Y :	REAL;
	END_VAR

	IF X > 0.0 THEN
		ATAN2 := ATAN(Y/X);
	ELSIF X < 0.0 THEN
		IF Y >= 0.0 THEN
			ATAN2 := ATAN(Y/X) + 3.14159265358979323846264338327950288;
		ELSE
			ATAN2 := ATAN(Y/X) - 3.14159265358979323846264338327950288;
		END_IF;
	ELSIF Y > 0.0 THEN
		ATAN2 := 1.5707963267948965580;
	ELSIF Y < 0.0 THEN
		ATAN2 := -1.5707963267948965580;
	ELSE
		ATAN2 := 0.0;
	END_IF;

END_FUNCTION

FUNCTION HYPOT:REAL
	VAR_INPUT
		X :	REAL;
		Y :	REAL;
	END_VAR

	HYPOT := SQRT(x*x + y*y);
END_FUNCTION

FUNCTION_BLOCK CLOG_Block

	VAR_INPUT
		X :	oscat_complex;
	END_VAR

	VAR_OUTPUT
		CLOG :	oscat_complex;
	END_VAR

	CLOG.re := LN(HYPOT(X.re, X.im));
	CLOG.im := ATAN2(X.im, X.re);

END_FUNCTION_BLOCK

FUNCTION_BLOCK CPOW_Block
	VAR_INPUT
		X :	oscat_complex;
		Y :	oscat_complex;
	END_VAR

	VAR_OUTPUT
		CPOW :	oscat_complex;
	END_VAR

	VAR
		CLOG :	CLOG_Block;
		CEXP :	CEXP_Block;
		CMUL :	CMUL_Block;
	END_VAR

	CLOG(X:=X);
	CMUL(X:=Y,Y:=CLOG.CLOG);
	CEXP(X:=CMUL.CMUL);
	CPOW := CEXP.CEXP;
END_FUNCTION_BLOCK

PROGRAM program0
  VAR
    LocalVar0 : oscat_complex;
	LocalVar1 : oscat_complex;
	LocalOUT  : oscat_complex;
	func_block : CPOW_Block;
  END_VAR
	func_block.X  := LocalVar0;
	func_block.Y  := LocalVar1;
	func_block();
	LocalOUT := func_block.CPOW;
END_PROGRAM

CONFIGURATION Config0
  RESOURCE Res0 ON PLC
    TASK task0(INTERVAL := T#20ms,PRIORITY := 0);
    PROGRAM instance0 WITH task0 : program0;
  END_RESOURCE
END_CONFIGURATION

(* ---- CRC_GEN.ST ---- *)
TYPE
	oscat_arb_0_249 			  : ARRAY [0..249] 	OF BYTE;
END_TYPE

FUNCTION REVERSE:BYTE
VAR_INPUT
	IN :	BYTE;
END_VAR

reverse := SHL(in,7) OR SHR(in,7) OR (ROR(in,3) AND BYTE#2#01000100) OR (ROL(in,3) AND BYTE#2#00100010)
	OR (SHL(in,1) AND BYTE#2#00010000) OR (SHR(in,1) AND BYTE#2#00001000);

END_FUNCTION

FUNCTION REFLECT:DWORD
	VAR_INPUT
		D :	DWORD;
		L :	INT;
	END_VAR

	VAR
		i :	INT;
		_d :	DWORD;
	END_VAR

	REFLECT := DWORD#0;
	_d := D;
	FOR i := 1 TO L DO
		REFLECT := SHL(REFLECT, 1) OR BOOL_TO_DWORD((_d AND DWORD#2#0000_0001) > DWORD#0); (* D.0 *)
		_d := SHR(_d, 1);
	END_FOR;
	REFLECT := REFLECT OR SHL(_d, L);
END_FUNCTION

FUNCTION_BLOCK CRC_GEN_Block
	VAR_IN_OUT
		PT :	oscat_arb_0_249;
	END_VAR

	VAR_INPUT
		SIZE :	UINT;
		PL :	UINT;
		PN :	DWORD;
		INIT :	DWORD;
		REV_IN :	BOOL;
		REV_OUT :	BOOL;
		XOR_OUT :	DWORD;
	END_VAR

	VAR_OUTPUT
		CRC_GEN :	DWORD;
	END_VAR

	VAR
		pos :	INT;
		shift :	INT;
		dx :	BYTE;
		bits :	INT;
	END_VAR

	shift := 32 - UINT_TO_INT(PL);
	PN := SHL(PN, shift);

	FOR pos := 0 TO 3 DO
		IF REV_IN THEN CRC_GEN := SHL(CRC_GEN, 8) OR BYTE_TO_DWORD(REVERSE(PT[pos])); ELSE CRC_GEN := SHL(CRC_GEN, 8) OR BYTE_TO_DWORD(PT[pos]); END_IF;
	END_FOR;
	pos := 4;

	CRC_GEN := CRC_GEN XOR SHL(init, shift);

	WHILE pos < UINT_TO_INT(size) DO
		IF REV_IN THEN DX := REVERSE(PT[pos]); ELSE DX := PT[pos]; END_IF;
		pos := pos + 1;
		FOR bits := 0 TO 7 DO
			IF (CRC_GEN AND DWORD#16#8000_0000) > DWORD#0 THEN (* CRC_GEN.31 *)
				CRC_GEN := (SHL(CRC_GEN, 1) OR BOOL_TO_DWORD((DX AND BYTE#16#80) > BYTE#0)) XOR PN; (* DX.7 *)
			ELSE
				CRC_GEN := SHL(CRC_GEN, 1) OR BOOL_TO_DWORD((DX AND BYTE#16#80) > BYTE#0); (* DX.7 *)
			END_IF;
			dx := SHL(dx, 1);
		END_FOR;
	END_WHILE;

	FOR bits := 0 TO 31 DO
		IF (CRC_GEN AND DWORD#16#8000_0000) > DWORD#0 THEN (* CRC_GEN.31 *)
			CRC_GEN := (SHL(CRC_GEN, 1) OR BOOL_TO_DWORD((DX AND BYTE#16#80) > BYTE#0)) XOR PN; (* DX.7 *)
		ELSE
			CRC_GEN := SHL(CRC_GEN, 1) OR BOOL_TO_DWORD((DX AND BYTE#16#80) > BYTE#0); (* DX.7 *)
		END_IF;
	END_FOR;

	CRC_GEN := SHR(CRC_GEN, shift) XOR XOR_OUT;

	IF REV_OUT THEN CRC_GEN := REFLECT(CRC_GEN, UINT_TO_INT(PL)); END_IF;

END_FUNCTION_BLOCK

PROGRAM program0
  VAR
	PT :	oscat_arb_0_249;

	SIZE :	UINT;
	PL :	UINT;
	PN :	DWORD;
	INIT :	DWORD;
	REV_IN :	BOOL;
	REV_OUT :	BOOL;
	XOR_OUT :	DWORD;

	CRC_GEN :	DWORD;
	func_block : CRC_GEN_Block;
  END_VAR
	func_block.PT  :=PT ;
	func_block.SIZE  :=SIZE ;
	func_block.PL  :=PL ;
	func_block.PN  :=PN ;
	func_block.INIT  :=INIT ;
	func_block.REV_IN  :=REV_IN ;
	func_block.REV_OUT  :=REV_OUT ;
	func_block.XOR_OUT  :=XOR_OUT ;
	func_block();

	PT := func_block.PT;
	CRC_GEN := func_block.CRC_GEN;
END_PROGRAM

CONFIGURATION Config0
  RESOURCE Res0 ON PLC
    TASK task0(INTERVAL := T#20ms,PRIORITY := 0);
    PROGRAM instance0 WITH task0 : program0;
  END_RESOURCE
END_CONFIGURATION

(* ---- CSET.ST ---- *)
TYPE oscat_complex :
  STRUCT
	re : REAL;
	im : REAL;
  END_STRUCT;
END_TYPE

FUNCTION_BLOCK CSET_Block
	VAR_INPUT
		RE :	REAL;
		IM :	REAL;
	END_VAR

	VAR_OUTPUT
		CSET :	oscat_complex;
	END_VAR

	CSET.re := RE;
	CSET.im := IM;
END_FUNCTION_BLOCK

PROGRAM program0
  VAR
    LocalVar0 : REAL;
	LocalVar1 : REAL;
	LocalOUT  : oscat_complex;
	func_block : CSET_Block;
  END_VAR
	func_block.RE  := LocalVar0;
	func_block.IM  := LocalVar1;
	func_block();
	LocalOUT := func_block.CSET;
END_PROGRAM

CONFIGURATION Config0
  RESOURCE Res0 ON PLC
    TASK task0(INTERVAL := T#20ms,PRIORITY := 0);
    PROGRAM instance0 WITH task0 : program0;
  END_RESOURCE
END_CONFIGURATION

(* ---- CSIN.ST ---- *)
TYPE oscat_complex :
  STRUCT
	re : REAL;
	im : REAL;
  END_STRUCT;
END_TYPE

FUNCTION COSH:REAL
	VAR_INPUT
		X :	REAL;
	END_VAR

	VAR
		t :	REAL;
	END_VAR

	T := EXP(X);
	COSH := (1.0 / T + T) * 0.5;
END_FUNCTION

FUNCTION SINH:REAL
	VAR_INPUT
		X :	REAL;
	END_VAR

	IF ABS(x) < 2.0E-3 THEN
		SINH := X;
	ELSE
		SINH := (EXP(x) - EXP(-x)) * 0.5;
	END_IF;
END_FUNCTION

FUNCTION_BLOCK CSIN_Block
	VAR_INPUT
		X :	oscat_complex;
	END_VAR

	VAR_OUTPUT
		CSIN :	oscat_complex;
	END_VAR

	CSIN.re := cosH(X.im) * SIN(X.re);
	CSIN.im := sinH(X.im) * COS(X.re);
END_FUNCTION_BLOCK

PROGRAM program0
  VAR
    LocalVar0 : oscat_complex;
	LocalOUT  : oscat_complex;
	func_block : CSIN_Block;
  END_VAR
	func_block.X  := LocalVar0;
	func_block();
	LocalOUT := func_block.CSIN;
END_PROGRAM

CONFIGURATION Config0
  RESOURCE Res0 ON PLC
    TASK task0(INTERVAL := T#20ms,PRIORITY := 0);
    PROGRAM instance0 WITH task0 : program0;
  END_RESOURCE
END_CONFIGURATION

(* ---- CSINH.ST ---- *)
TYPE oscat_complex :
  STRUCT
	re : REAL;
	im : REAL;
  END_STRUCT;
END_TYPE

FUNCTION COSH:REAL
	VAR_INPUT
		X :	REAL;
	END_VAR

	VAR
		t :	REAL;
	END_VAR

	T := EXP(X);
	COSH := (1.0 / T + T) * 0.5;
END_FUNCTION

FUNCTION SINH:REAL
	VAR_INPUT
		X :	REAL;
	END_VAR

	IF ABS(x) < 2.0E-3 THEN
		SINH := X;
	ELSE
		SINH := (EXP(x) - EXP(-x)) * 0.5;
	END_IF;
END_FUNCTION

FUNCTION_BLOCK CSINH_Block

	VAR_INPUT
		X :	oscat_complex;
	END_VAR

	VAR_OUTPUT
		CSINH :	oscat_complex;
	END_VAR

	CSINH.re := sinH(X.re) * COS(X.im);
	CSINH.im := cosH(X.re) * SIN(X.im);

END_FUNCTION_BLOCK

PROGRAM program0
  VAR
    LocalVar0 : oscat_complex;
	LocalOUT  : oscat_complex;
	func_block : CSINH_Block;
  END_VAR
	func_block.X  := LocalVar0;
	func_block();
	LocalOUT := func_block.CSINH;
END_PROGRAM

CONFIGURATION Config0
  RESOURCE Res0 ON PLC
    TASK task0(INTERVAL := T#20ms,PRIORITY := 0);
    PROGRAM instance0 WITH task0 : program0;
  END_RESOURCE
END_CONFIGURATION

(* ---- CSQRT.ST ---- *)
TYPE oscat_complex :
  STRUCT
	re : REAL;
	im : REAL;
  END_STRUCT;
END_TYPE

FUNCTION HYPOT:REAL
	VAR_INPUT
		X :	REAL;
		Y :	REAL;
	END_VAR

	HYPOT := SQRT(x*x + y*y);
END_FUNCTION

FUNCTION SGN : INT
  VAR_INPUT
    x : REAL;
  END_VAR

  IF X > 0.0 THEN
  	sgn := 1;
  ELSIF X < 0.0 THEN
  	sgn := -1;
  ELSE
  	sgn := 0;
  END_IF;
END_FUNCTION

FUNCTION_BLOCK CSQRT_Block
	VAR_INPUT
		X :	oscat_complex;
	END_VAR

	VAR_OUTPUT
		CSQRT :	oscat_complex;
	END_VAR

	VAR
		temp :	REAL;
	END_VAR

	temp := HYPOT(x.re, x.im);
	CSQRT.re :=  SQRT(0.5 * (temp + x.re));
	CSQRT.im :=  INT_TO_REAL(sgn(x.im)) * SQRT(0.5 * (temp - x.re));

END_FUNCTION_BLOCK

PROGRAM program0
  VAR
    LocalVar0 : oscat_complex;
	LocalOUT  : oscat_complex;
	func_block : CSQRT_Block;
  END_VAR
	func_block.X  := LocalVar0;
	func_block();
	LocalOUT := func_block.CSQRT;
END_PROGRAM

CONFIGURATION Config0
  RESOURCE Res0 ON PLC
    TASK task0(INTERVAL := T#20ms,PRIORITY := 0);
    PROGRAM instance0 WITH task0 : program0;
  END_RESOURCE
END_CONFIGURATION

(* ---- CSUB.ST ---- *)
TYPE oscat_complex :
  STRUCT
	re : REAL;
	im : REAL;
  END_STRUCT;
END_TYPE

FUNCTION_BLOCK CSUB_Block
	VAR_INPUT
		X :	oscat_complex;
		Y :	oscat_complex;
	END_VAR

	VAR_OUTPUT
		CSUB :	oscat_complex;
	END_VAR

	CSUB.re := X.re - Y.re;
	CSUB.im := X.im - Y.im;
END_FUNCTION_BLOCK

PROGRAM program0
  VAR
    LocalVar0 : oscat_complex;
	LocalVar1 : oscat_complex;
	LocalOUT  : oscat_complex;
	func_block : CSUB_Block;
  END_VAR
	func_block.X  := LocalVar0;
	func_block.Y  := LocalVar0;
	func_block();
	LocalOUT := func_block.CSUB;
END_PROGRAM

CONFIGURATION Config0
  RESOURCE Res0 ON PLC
    TASK task0(INTERVAL := T#20ms,PRIORITY := 0);
    PROGRAM instance0 WITH task0 : program0;
  END_RESOURCE
END_CONFIGURATION

(* ---- CTAN.ST ---- *)
TYPE oscat_complex :
  STRUCT
	re : REAL;
	im : REAL;
  END_STRUCT;
END_TYPE

FUNCTION COSH:REAL
	VAR_INPUT
		X :	REAL;
	END_VAR

	VAR
		t :	REAL;
	END_VAR

	T := EXP(X);
	COSH := (1.0 / T + T) * 0.5;
END_FUNCTION

FUNCTION SINH:REAL
	VAR_INPUT
		X :	REAL;
	END_VAR

	IF ABS(x) < 2.0E-3 THEN
		SINH := X;
	ELSE
		SINH := (EXP(x) - EXP(-x)) * 0.5;
	END_IF;
END_FUNCTION

FUNCTION_BLOCK CTAN_Block
	VAR_INPUT
		X :	oscat_complex;
	END_VAR

	VAR_OUTPUT
		CTAN :	oscat_complex;
	END_VAR

	VAR
		temp :	REAL;
		xi2 :	REAL;
		xr2 :	REAL;
	END_VAR

	xi2 := 2.0 * x.im;
	xr2 := 2.0 * x.re;
	temp := 1.0 / (COS(xr2) + COSH( xi2));
	CTAN.re := temp * SIN(xr2);
	CTAN.im := temp * SINH(xi2);
END_FUNCTION_BLOCK

PROGRAM program0
  VAR
    LocalVar0 : oscat_complex;
	LocalOUT  : oscat_complex;
	func_block : CTAN_Block;
  END_VAR
	func_block.X  := LocalVar0;
	func_block();
	LocalOUT := func_block.CTAN;
END_PROGRAM

CONFIGURATION Config0
  RESOURCE Res0 ON PLC
    TASK task0(INTERVAL := T#20ms,PRIORITY := 0);
    PROGRAM instance0 WITH task0 : program0;
  END_RESOURCE
END_CONFIGURATION

(* ---- CTANH.ST ---- *)
TYPE oscat_complex :
  STRUCT
	re : REAL;
	im : REAL;
  END_STRUCT;
END_TYPE

FUNCTION COSH:REAL
	VAR_INPUT
		X :	REAL;
	END_VAR

	VAR
		t :	REAL;
	END_VAR

	T := EXP(X);
	COSH := (1.0 / T + T) * 0.5;
END_FUNCTION

FUNCTION SINH:REAL
	VAR_INPUT
		X :	REAL;
	END_VAR

	IF ABS(x) < 2.0E-3 THEN
		SINH := X;
	ELSE
		SINH := (EXP(x) - EXP(-x)) * 0.5;
	END_IF;
END_FUNCTION

FUNCTION_BLOCK CTANH_Block
	VAR_INPUT
		X :	oscat_complex;
	END_VAR

	VAR_OUTPUT
		CTANH :	oscat_complex;
	END_VAR

	VAR
		xi2 :	REAL;
		xr2 :	REAL;
		temp :	REAL;
	END_VAR

	xi2 := 2.0 * x.im;
	xr2 := 2.0 * x.re;
	temp := 1.0 /(COSH(xr2) + COS(xi2));
	CTANH.re := temp * SINH(xr2);
	CTANH.im := temp * SIN(xi2);

END_FUNCTION_BLOCK

PROGRAM program0
  VAR
    LocalVar0 : oscat_complex;
	LocalOUT  : oscat_complex;
	func_block : CTANH_Block;
  END_VAR
	func_block.X  := LocalVar0;
	func_block();
	LocalOUT := func_block.CTANH;
END_PROGRAM

CONFIGURATION Config0
  RESOURCE Res0 ON PLC
    TASK task0(INTERVAL := T#20ms,PRIORITY := 0);
    PROGRAM instance0 WITH task0 : program0;
  END_RESOURCE
END_CONFIGURATION

(* ---- CTRL_OUT.ST ---- *)
FUNCTION_BLOCK CTRL_OUT
	VAR_INPUT
		CI :	REAL;
		OFFSET :	REAL;
		MAN_IN :	REAL;
		LIM_L :	REAL;
		LIM_H :	REAL;
		MANUAL :	BOOL;
	END_VAR

	VAR_OUTPUT
		Y :	REAL;
		LIM :	BOOL;
	END_VAR

	Y := SEL(manual, CI, MAN_IN) + OFFSET;

	IF Y >= LIM_H THEN
		Y := LIM_H;
		LIM := TRUE;
	ELSIF Y <= lim_L THEN
		Y := LIM_L;
		LIM := TRUE;
	ELSE
		LIM := FALSE;
	END_IF;
END_FUNCTION_BLOCK

PROGRAM program0
  VAR
	CI :	REAL;
	OFFSET :	REAL;
	MAN_IN :	REAL;
	LIM_L :	REAL;
	LIM_H :	REAL;
	MANUAL :	BOOL;

	Y :	REAL;
	LIM :	BOOL;

	func_block : CTRL_OUT;
  END_VAR
	func_block.CI  := CI ;
	func_block.OFFSET   :=OFFSET ;
	func_block.MAN_IN   :=MAN_IN ;
	func_block.LIM_L   :=LIM_L ;
	func_block.LIM_H   :=LIM_H ;
	func_block.MANUAL   :=MANUAL ;
	func_block();
	Y := func_block.Y;
	LIM := func_block.LIM;
END_PROGRAM

CONFIGURATION Config0
  RESOURCE Res0 ON PLC
    TASK task0(INTERVAL := T#20ms,PRIORITY := 0);
    PROGRAM instance0 WITH task0 : program0;
  END_RESOURCE
END_CONFIGURATION

(* ---- CTRL_PI.ST ---- *)
FUNCTION_BLOCK T_PLC_US_Block
	VAR_OUTPUT
		T_PLC_US :	UDINT;
	END_VAR

	VAR_EXTERNAL
		PLC_TICKS_PER_SEC :	INT;
		PLC_SYS_TICK_CNT :	DINT;
	END_VAR

	VAR
		debug :	BOOL;
		N :	INT;
		Offset :	UDINT;
		temp :	DWORD := DWORD#1;
		mode :	BOOL;
		faktor :	UDINT;
		init :	BOOL;
		v_plc_ticks_per_sec :	UDINT;
		base :	UDINT := UDINT#1000000;
	END_VAR

	IF init = FALSE THEN
		v_plc_ticks_per_sec := INT_TO_UDINT(PLC_TICKS_PER_SEC);
		IF v_plc_ticks_per_sec = UDINT#1024 THEN
			faktor := UDINT#1000;
			mode := FALSE;
		ELSIF v_plc_ticks_per_sec > UDINT#0 THEN
			IF v_plc_ticks_per_sec <= base THEN
				faktor := base / v_plc_ticks_per_sec;
				mode := FALSE;
			ELSE
				faktor := v_plc_ticks_per_sec / base;
				mode := TRUE;
			END_IF;
		ELSE
			faktor := UDINT#1;
		END_IF;
		init := TRUE;
	END_IF;

	IF mode THEN
		T_PLC_US := DINT_TO_UDINT(PLC_SYS_TICK_CNT) / faktor;
	ELSE
		T_PLC_US := DINT_TO_UDINT(PLC_SYS_TICK_CNT) * faktor;
	END_IF;

	IF debug THEN
		T_PLC_US := (DWORD_TO_UDINT(SHL(UDINT_TO_DWORD(T_PLC_US),N) OR SHL(temp,N)) - UDINT#1) + Offset;
	END_IF;
END_FUNCTION_BLOCK

FUNCTION_BLOCK FT_PIWL

	VAR_INPUT
		IN :	REAL;
		KP :	REAL := 1.0;
		KI :	REAL := 1.0;
		LIM_L :	REAL := -1.0E38;
		LIM_H :	REAL := 1.0E38;
		RST :	BOOL;
	END_VAR

	VAR_OUTPUT
		Y :	REAL;
		LIM :	BOOL;
	END_VAR

	VAR
		init :	BOOL;
		tx :	UDINT;
		tc :	REAL;
		t_last :	UDINT;
		in_last :	REAL;
		i :	REAL;
		p :	REAL;
		T_PLC_US :	T_PLC_US_Block;
	END_VAR

	IF NOT init OR RST THEN
		init := TRUE;
		in_last := in;
		T_PLC_US();
		t_last := T_PLC_US.T_PLC_US;
		i := 0.0;
		tc := 0.0;
	ELSE
		(* read last cycle time in Microseconds *)
		T_PLC_US();
		tx := T_PLC_US.T_PLC_US;
		tc := UDINT_TO_REAL(tx - t_last);
		t_last := tx;

		(* calculate proportional part *)
		p := KP * IN;

		(* run integrator *)
		i := (IN + in_last) * 5.0E-7 * KI * tc + i;
		in_last := IN;

		(* calculate output Y *)
		Y := p + i;

		(* check output for limits *)
		IF Y >= LIM_H THEN
			Y := LIM_H;
			IF ki <> 0.0 THEN
				i := LIM_H - p;
			ELSE
				i := 0.0;
			END_IF;
			LIM := TRUE;
		ELSIF Y <= LIM_L THEN
			Y := LIM_L;
			IF ki <> 0.0 THEN
				i := LIM_L - p;
			ELSE
				i := 0.0;
			END_IF;
			LIM := TRUE;
		ELSE
			LIM := FALSE;
		END_IF;
	END_IF;
END_FUNCTION_BLOCK

FUNCTION_BLOCK CTRL_OUT
	VAR_INPUT
		CI :	REAL;
		OFFSET :	REAL;
		MAN_IN :	REAL;
		LIM_L :	REAL;
		LIM_H :	REAL;
		MANUAL :	BOOL;
	END_VAR

	VAR_OUTPUT
		Y :	REAL;
		LIM :	BOOL;
	END_VAR

	Y := SEL(manual, CI, MAN_IN) + OFFSET;

	IF Y >= LIM_H THEN
		Y := LIM_H;
		LIM := TRUE;
	ELSIF Y <= lim_L THEN
		Y := LIM_L;
		LIM := TRUE;
	ELSE
		LIM := FALSE;
	END_IF;
END_FUNCTION_BLOCK

FUNCTION DEAD_ZONE:REAL

	VAR_INPUT
		X :	REAL;
		L :	REAL;
	END_VAR

	IF ABS(x) > L THEN
		dead_zone := X;
	ELSE
		DEAD_ZONE := 0.0;
	END_IF;

END_FUNCTION

FUNCTION CTRL_IN:REAL
	VAR_INPUT
		SET_POINT :	REAL;
		ACTUAL :	REAL;
		NOISE :	REAL;
	END_VAR
	CTRL_IN := DEAD_ZONE(SET_POINT - ACTUAL, NOISE);
END_FUNCTION

FUNCTION_BLOCK CTRL_PI
	VAR_INPUT
		ACT :	REAL;
		SET :	REAL;
		SUP :	REAL;
		OFS :	REAL;
		M_I :	REAL;
		MAN :	BOOL;
		RST :	BOOL := FALSE;
		KP  :	REAL := 1.0;
		KI  :	REAL := 1.0;
		LL  :	REAL := -1000.0;
		LH  :	REAL := 1000.0;
	END_VAR

	VAR_OUTPUT
		Y    :	REAL;
		DIFF :	REAL;
		LIM  :	BOOL;
	END_VAR

	VAR
		pi :	FT_PIWL;
		co :	CTRL_OUT;
	END_VAR

	DIFF := CTRL_IN(SET, ACT, SUP);
	pi(in := DIFF, kp := KP, ki := KI, lim_l := LL, lim_h := LH, rst := RST);
	co(ci := pi.Y, OFFSET := OFS, man_in := M_I, lim_l := LL, lim_h := LH, manual := MAN);
	Y := co.Y;
	LIM := co.LIM;
END_FUNCTION_BLOCK

PROGRAM program0
  VAR
		ACT :	REAL;
		SET :	REAL;
		SUP :	REAL;
		OFS :	REAL;
		M_I :	REAL;
		MAN :	BOOL;
		RST :	BOOL;
		KP  :	REAL;
		KI  :	REAL;
		LL  :	REAL;
		LH  :	REAL;

		Y    :	REAL;
		DIFF :	REAL;
		LIM  :	BOOL;

	func_block : CTRL_PI;
  END_VAR
	func_block.ACT  :=ACT ;
	func_block.SET  :=SET ;
	func_block.SUP  :=SUP ;
	func_block.OFS  :=OFS ;
	func_block.M_I  :=M_I ;
	func_block.MAN  :=MAN ;
	func_block.RST  :=RST ;
	func_block.KP   :=KP  ;
	func_block.KI   :=KI  ;
	func_block.LL   :=LL  ;
	func_block.LH   :=LH  ;

	func_block();
	Y    := func_block.Y   ;
	DIFF := func_block.DIFF;
	LIM  := func_block.LIM ;
END_PROGRAM

CONFIGURATION Config0
	VAR_GLOBAL
		PLC_TICKS_PER_SEC :	INT;
		PLC_SYS_TICK_CNT :	DINT;
	END_VAR

	RESOURCE Res0 ON PLC
		TASK task0(INTERVAL := T#20ms,PRIORITY := 0);
		PROGRAM instance0 WITH task0 : program0;
	END_RESOURCE
END_CONFIGURATION

(* ---- CTRL_PID.ST ---- *)
FUNCTION_BLOCK T_PLC_US_Block
	VAR_OUTPUT
		T_PLC_US :	UDINT;
	END_VAR

	VAR_EXTERNAL
		PLC_TICKS_PER_SEC :	INT;
		PLC_SYS_TICK_CNT :	DINT;
	END_VAR

	VAR
		debug :	BOOL;
		N :	INT;
		Offset :	UDINT;
		temp :	DWORD := DWORD#1;
		mode :	BOOL;
		faktor :	UDINT;
		init :	BOOL;
		v_plc_ticks_per_sec :	UDINT;
		base :	UDINT := UDINT#1000000;
	END_VAR

	IF init = FALSE THEN
		v_plc_ticks_per_sec := INT_TO_UDINT(PLC_TICKS_PER_SEC);
		IF v_plc_ticks_per_sec = UDINT#1024 THEN
			faktor := UDINT#1000;
			mode := FALSE;
		ELSIF v_plc_ticks_per_sec > UDINT#0 THEN
			IF v_plc_ticks_per_sec <= base THEN
				faktor := base / v_plc_ticks_per_sec;
				mode := FALSE;
			ELSE
				faktor := v_plc_ticks_per_sec / base;
				mode := TRUE;
			END_IF;
		ELSE
			faktor := UDINT#1;
		END_IF;
		init := TRUE;
	END_IF;

	IF mode THEN
		T_PLC_US := DINT_TO_UDINT(PLC_SYS_TICK_CNT) / faktor;
	ELSE
		T_PLC_US := DINT_TO_UDINT(PLC_SYS_TICK_CNT) * faktor;
	END_IF;

	IF debug THEN
		T_PLC_US := (DWORD_TO_UDINT(SHL(UDINT_TO_DWORD(T_PLC_US),N) OR SHL(temp,N)) - UDINT#1) + Offset;
	END_IF;
END_FUNCTION_BLOCK

FUNCTION_BLOCK FT_PIWL

	VAR_INPUT
		IN :	REAL;
		KP :	REAL := 1.0;
		KI :	REAL := 1.0;
		LIM_L :	REAL := -1.0E38;
		LIM_H :	REAL := 1.0E38;
		RST :	BOOL;
	END_VAR

	VAR_OUTPUT
		Y :	REAL;
		LIM :	BOOL;
	END_VAR

	VAR
		init :	BOOL;
		tx :	UDINT;
		tc :	REAL;
		t_last :	UDINT;
		in_last :	REAL;
		i :	REAL;
		p :	REAL;
		T_PLC_US :	T_PLC_US_Block;
	END_VAR

	IF NOT init OR RST THEN
		init := TRUE;
		in_last := in;
		T_PLC_US();
		t_last := T_PLC_US.T_PLC_US;
		i := 0.0;
		tc := 0.0;
	ELSE
		(* read last cycle time in Microseconds *)
		T_PLC_US();
		tx := T_PLC_US.T_PLC_US;
		tc := UDINT_TO_REAL(tx - t_last);
		t_last := tx;

		(* calculate proportional part *)
		p := KP * IN;

		(* run integrator *)
		i := (IN + in_last) * 5.0E-7 * KI * tc + i;
		in_last := IN;

		(* calculate output Y *)
		Y := p + i;

		(* check output for limits *)
		IF Y >= LIM_H THEN
			Y := LIM_H;
			IF ki <> 0.0 THEN
				i := LIM_H - p;
			ELSE
				i := 0.0;
			END_IF;
			LIM := TRUE;
		ELSIF Y <= LIM_L THEN
			Y := LIM_L;
			IF ki <> 0.0 THEN
				i := LIM_L - p;
			ELSE
				i := 0.0;
			END_IF;
			LIM := TRUE;
		ELSE
			LIM := FALSE;
		END_IF;
	END_IF;
END_FUNCTION_BLOCK

FUNCTION_BLOCK FT_DERIV
	VAR_INPUT
		IN :	REAL;
		K :	REAL := 1.0;
		RUN :	BOOL := TRUE;
	END_VAR

	VAR_OUTPUT
		OUT :	REAL;
	END_VAR

	VAR
		old :	REAL;
		tx :	UDINT;
		last :	UDINT;
		init :	BOOL;
		tc :	REAL;
		T_PLC_US :	T_PLC_US_Block;
	END_VAR

	T_PLC_US();
	tx:= T_PLC_US.T_PLC_US;
	tc := UDINT_TO_REAL(tx - last);

	IF NOT init THEN
		init := TRUE;
		old := in;
	ELSIF run AND tc > 0.0 THEN
		out := (in - old) / tc * 1000000.0 * K;
		old := in;
	ELSE
		out := 0.0;
	END_IF;

	last := tx;

	T_PLC_US();
	tx:= T_PLC_US.T_PLC_US;

	IF NOT init THEN
		init := TRUE;
	ELSIF run AND tx - last > UDINT#0 THEN
		out := (in - old) / UDINT_TO_REAL(tx - last) * 1000000.0 * K;
	ELSE
		out := 0.0;
	END_IF;
	old := in;
	last := tx;
END_FUNCTION_BLOCK

FUNCTION_BLOCK FT_PIDWL
	VAR_INPUT
		IN :	REAL;
		KP :	REAL := 1.0;
		TN :	REAL := 1.0;
		TV :	REAL := 1.0;
		LIM_L :	REAL := -1.0E38;
		LIM_H :	REAL := 1.0E38;
		RST :	BOOL;
	END_VAR

	VAR_OUTPUT
		Y :	REAL;
		LIM :	BOOL;
	END_VAR

	VAR
		piwl :	FT_PIWL;
		diff :	FT_DERIV;
	END_VAR

	IF rst THEN
		piwl(rst := TRUE);
		piwl.RST := FALSE;
	ELSE
		IF TN = 0.0 THEN
			piwl(in := IN * KP, KP := 1.0, KI := 0.0, LIM_L := LIM_L, LIM_H := LIM_H);
		ELSE
			piwl(in := IN * KP, KP := 1.0, KI := 1.0 / TN, LIM_L := LIM_L, LIM_H := LIM_H);
		END_IF;

		diff(IN := IN, K := KP * TV);
		Y := piwl.Y + diff.out;

		IF Y < LIM_L THEN
			LIM := TRUE;
			Y := LIM_L;
		ELSIF Y > LIM_H THEN
			LIM := TRUE;
			Y := LIM_H;
		ELSE
			LIM := FALSE;
		END_IF;
	END_IF;
END_FUNCTION_BLOCK

FUNCTION_BLOCK CTRL_OUT
	VAR_INPUT
		CI :	REAL;
		OFFSET :	REAL;
		MAN_IN :	REAL;
		LIM_L :	REAL;
		LIM_H :	REAL;
		MANUAL :	BOOL;
	END_VAR

	VAR_OUTPUT
		Y :	REAL;
		LIM :	BOOL;
	END_VAR

	Y := SEL(manual, CI, MAN_IN) + OFFSET;

	IF Y >= LIM_H THEN
		Y := LIM_H;
		LIM := TRUE;
	ELSIF Y <= lim_L THEN
		Y := LIM_L;
		LIM := TRUE;
	ELSE
		LIM := FALSE;
	END_IF;
END_FUNCTION_BLOCK

FUNCTION DEAD_ZONE:REAL

	VAR_INPUT
		X :	REAL;
		L :	REAL;
	END_VAR

	IF ABS(x) > L THEN
		dead_zone := X;
	ELSE
		DEAD_ZONE := 0.0;
	END_IF;

END_FUNCTION

FUNCTION CTRL_IN:REAL
	VAR_INPUT
		SET_POINT :	REAL;
		ACTUAL :	REAL;
		NOISE :	REAL;
	END_VAR
	CTRL_IN := DEAD_ZONE(SET_POINT - ACTUAL, NOISE);
END_FUNCTION

FUNCTION_BLOCK CTRL_PID
	VAR_INPUT
		ACT :	REAL;
		SET :	REAL;
		SUP :	REAL;
		OFS :	REAL;
		M_I :	REAL;
		MAN :	BOOL;
		RST :	BOOL := FALSE;
		KP :	REAL := 1.0;
		TN :	REAL := 1.0;
		TV :	REAL := 1.0;
		LL :	REAL := -1000.0;
		LH :	REAL := 1000.0;
	END_VAR

	VAR_OUTPUT
		Y :	REAL;
		DIFF :	REAL;
		LIM :	BOOL;
	END_VAR

	VAR
		pidd :	FT_PIDWL;
		co :	CTRL_OUT;
	END_VAR

	DIFF := CTRL_IN(SET, ACT, SUP);
	pidd(in := DIFF, kp := KP, tn := TN, tv := TV, lim_l := LL, lim_h := LH, rst := RST);
	co(ci := pidd.Y, OFFSET := OFS, man_in := M_I, lim_l := LL, lim_h := LH, manual := MAN);
	Y := co.Y;
	LIM := co.LIM;
END_FUNCTION_BLOCK

PROGRAM program0
  VAR
		ACT :	REAL;
		SET :	REAL;
		SUP :	REAL;
		OFS :	REAL;
		M_I :	REAL;
		MAN :	BOOL;
		RST :	BOOL;
		KP :	REAL;
		TN  :	REAL;
		TV  :	REAL;
		LL  :	REAL;
		LH  :	REAL;

		Y    :	REAL;
		DIFF :	REAL;
		LIM  :	BOOL;

	func_block : CTRL_PID;
  END_VAR
	func_block.ACT  :=ACT ;
	func_block.SET  :=SET ;
	func_block.SUP  :=SUP ;
	func_block.OFS  :=OFS ;
	func_block.M_I  :=M_I ;
	func_block.MAN  :=MAN ;
	func_block.RST  :=RST ;
	func_block.KP   :=KP  ;
	func_block.TV   :=TV  ;
	func_block.TN   :=TN  ;
	func_block.LL   :=LL  ;
	func_block.LH   :=LH  ;

	func_block();
	Y    := func_block.Y   ;
	DIFF := func_block.DIFF;
	LIM  := func_block.LIM ;
END_PROGRAM

CONFIGURATION Config0
	VAR_GLOBAL
		PLC_TICKS_PER_SEC :	INT;
		PLC_SYS_TICK_CNT :	DINT;
	END_VAR

	RESOURCE Res0 ON PLC
		TASK task0(INTERVAL := T#20ms,PRIORITY := 0);
		PROGRAM instance0 WITH task0 : program0;
	END_RESOURCE
END_CONFIGURATION

(* ---- CTRL_PWM.ST ---- *)
FUNCTION_BLOCK T_PLC_MS_block
	VAR_OUTPUT
		T_PLC_MS :	UDINT;
	END_VAR

	VAR_EXTERNAL
		PLC_TICKS_PER_SEC :	INT;
		PLC_SYS_TICK_CNT :	DINT;
	END_VAR

	VAR
		debug :	BOOL;(*Debug-Mode ON / OFF*)
		N :	INT;(*Debug-Faktor*)
		Offset :	UDINT;(*Debug-Offset*)
		temp :	DWORD := DWORD#1;(*Debug-Offset*)
		mode :	BOOL;(*modus*)
		faktor :	UDINT;(*Systemtakt-Faktor*)
		init :	BOOL;
		v_plc_ticks_per_sec :	UDINT;
		base :	UDINT := UDINT#1000;
	END_VAR

	IF init = FALSE THEN
		v_plc_ticks_per_sec := INT_TO_UDINT(PLC_TICKS_PER_SEC);
		IF v_plc_ticks_per_sec = UDINT#1024 THEN
			faktor := UDINT#1;
			mode := FALSE;
		ELSIF v_plc_ticks_per_sec > UDINT#0 THEN
			IF v_plc_ticks_per_sec <= base THEN
				faktor := base / v_plc_ticks_per_sec;
				mode := FALSE;
			ELSE
				faktor := v_plc_ticks_per_sec / base;
				mode := TRUE;
			END_IF;
		ELSE
			faktor := UDINT#1;
		END_IF;
		init := TRUE;
	END_IF;

	IF mode THEN
		T_PLC_MS := DINT_TO_UDINT(PLC_SYS_TICK_CNT) / faktor;
	ELSE
		T_PLC_MS := DINT_TO_UDINT(PLC_SYS_TICK_CNT) * faktor;
	END_IF;

	IF debug THEN
		T_PLC_MS := (DWORD_TO_UDINT(SHL(UDINT_TO_DWORD(T_PLC_MS),N) OR SHL(temp,N)) - UDINT#1) + Offset;
	END_IF;

END_FUNCTION_BLOCK

FUNCTION_BLOCK CLK_PRG
	VAR_INPUT
		PT :	TIME := T#10ms;
	END_VAR

	VAR_OUTPUT
		Q :	BOOL;
	END_VAR

	VAR
		init :	BOOL := FALSE;
		last :	TIME;
		tx :	TIME;
		T_PLC_MS :	T_PLC_MS_block;
	END_VAR

	T_PLC_MS();
	tx:= UDINT_TO_TIME(T_PLC_MS.T_PLC_MS);

	IF NOT init THEN
		init := TRUE;
		last := tx - pt;
	END_IF;

	Q := tx - last >= pt;
	IF Q THEN last := tx; END_IF;
END_FUNCTION_BLOCK

FUNCTION _REAL_TO_UDINT:UDINT
  VAR_INPUT
    X :	REAL;
  END_VAR

  IF REAL_TO_UDINT(0.5) = UDINT#1 THEN
    _REAL_TO_UDINT := REAL_TO_UDINT(x);
  ELSIF X > 0.0 THEN
    _REAL_TO_UDINT := REAL_TO_UDINT(x+0.5);
  ELSIF X < 0.0 THEN
    _REAL_TO_UDINT := REAL_TO_UDINT(x-0.5);
  ELSE
    _REAL_TO_UDINT := UDINT#0;
  END_IF;
END_FUNCTION

FUNCTION REAL_TO_TIME2:TIME
	VAR_INPUT
		IN :	REAL;
	END_VAR

	REAL_TO_TIME2 := DINT_TO_TIME(UDINT_TO_DINT(_REAL_TO_UDINT(IN)));
END_FUNCTION

FUNCTION_BLOCK TP_X
	VAR_INPUT
		IN :	BOOL;
		PT :	TIME;
	END_VAR

	VAR_OUTPUT
		Q :	BOOL;
		ET :	TIME;
	END_VAR

	VAR
		edge :	BOOL;
		start :	TIME;
		tx :	TIME;
		T_PLC_MS :	T_PLC_MS_block;
	END_VAR

	T_PLC_MS();
	tx := UDINT_TO_TIME(T_PLC_MS.T_PLC_MS);

	IF IN AND NOT edge THEN
		start := tx;
		Q := PT > t#0ms;
	ELSIF Q THEN
		ET := tx - start;
		IF ET >= PT THEN
			Q := FALSE;
			ET := t#0ms;
		END_IF;
	END_IF;
	edge := IN;

END_FUNCTION_BLOCK

FUNCTION_BLOCK PWM_DC
	VAR_INPUT
		F :	REAL;
		DC :	REAL;
	END_VAR

	VAR_OUTPUT
		Q :	BOOL;
	END_VAR

	VAR
		clk :	CLK_Prg;
		pulse :	TP_X;
		tmp :	REAL;
	END_VAR

	IF F > 0.0 THEN
		tmp := 1000.0/F;
		CLK(PT := REAL_TO_TIME2(tmp));
		Pulse(in := clk.Q, pt := REAL_TO_TIME2(tmp*DC));
		Q := pulse.Q;
	END_IF;
END_FUNCTION_BLOCK

FUNCTION_BLOCK CTRL_PWM
	VAR_INPUT
		CI :	REAL;
		MAN_IN :	REAL;
		MANUAL :	BOOL;
		F :	REAL;
	END_VAR

	VAR_OUTPUT
		Q :	BOOL;
	END_VAR

	VAR
		PW :	PWM_DC;
	END_VAR

	PW(F := F, DC := SEL(MANUAL,CI,MAN_IN));
	Q := PW.Q;
END_FUNCTION_BLOCK

PROGRAM program0
  VAR
	CI     :	REAL;
	MAN_IN :	REAL;
	MANUAL :	BOOL;
	F      :	REAL;

	Q :	BOOL;

	func_block : CTRL_PWM;
  END_VAR
	func_block.CI    :=CI    ;
	func_block.MAN_IN:=MAN_IN;
	func_block.MANUAL:=MANUAL;
	func_block.F     :=F     ;
	func_block();
	Q := func_block.Q;
END_PROGRAM

CONFIGURATION Config0
	VAR_GLOBAL
		PLC_TICKS_PER_SEC :	INT;
		PLC_SYS_TICK_CNT :	DINT;
	END_VAR

  RESOURCE Res0 ON PLC
    TASK task0(INTERVAL := T#20ms,PRIORITY := 0);
    PROGRAM instance0 WITH task0 : program0;
  END_RESOURCE
END_CONFIGURATION

(* ---- CYCLE_4.ST ---- *)
FUNCTION_BLOCK T_PLC_MS_block
	VAR_OUTPUT
		T_PLC_MS :	UDINT;
	END_VAR

	VAR_EXTERNAL
		PLC_TICKS_PER_SEC :	INT;
		PLC_SYS_TICK_CNT :	DINT;
	END_VAR

	VAR
		debug :	BOOL;(*Debug-Mode ON / OFF*)
		N :	INT;(*Debug-Faktor*)
		Offset :	UDINT;(*Debug-Offset*)
		temp :	DWORD := DWORD#1;(*Debug-Offset*)
		mode :	BOOL;(*modus*)
		faktor :	UDINT;(*Systemtakt-Faktor*)
		init :	BOOL;
		v_plc_ticks_per_sec :	UDINT;
		base :	UDINT := UDINT#1000;
	END_VAR

	IF init = FALSE THEN
		v_plc_ticks_per_sec := INT_TO_UDINT(PLC_TICKS_PER_SEC);
		IF v_plc_ticks_per_sec = UDINT#1024 THEN
			faktor := UDINT#1;
			mode := FALSE;
		ELSIF v_plc_ticks_per_sec > UDINT#0 THEN
			IF v_plc_ticks_per_sec <= base THEN
				faktor := base / v_plc_ticks_per_sec;
				mode := FALSE;
			ELSE
				faktor := v_plc_ticks_per_sec / base;
				mode := TRUE;
			END_IF;
		ELSE
			faktor := UDINT#1;
		END_IF;
		init := TRUE;
	END_IF;

	IF mode THEN
		T_PLC_MS := DINT_TO_UDINT(PLC_SYS_TICK_CNT) / faktor;
	ELSE
		T_PLC_MS := DINT_TO_UDINT(PLC_SYS_TICK_CNT) * faktor;
	END_IF;

	IF debug THEN
		T_PLC_MS := (DWORD_TO_UDINT(SHL(UDINT_TO_DWORD(T_PLC_MS),N) OR SHL(temp,N)) - UDINT#1) + Offset;
	END_IF;

END_FUNCTION_BLOCK

FUNCTION_BLOCK CYCLE_4

	VAR_INPUT
		E :	BOOL := TRUE;
		T0 :	TIME;
		T1 :	TIME;
		T2 :	TIME;
		T3 :	TIME;
		S0 :	BOOL;
		SX :	INT;
		SL :	BOOL;
	END_VAR

	VAR_OUTPUT
		STATE :	INT;
	END_VAR

	VAR
		tx :	TIME;
		last :	TIME;
		init :	BOOL;
		T_PLC_MS :	T_PLC_MS_block;
	END_VAR

	T_PLC_MS();
	tx:= UDINT_TO_TIME(T_PLC_MS.T_PLC_MS);

	(* init on first cycle *)
	IF NOT init THEN
		init := TRUE;
		last := tx;
	END_IF;

	IF E THEN
		IF SL THEN
			(* when sx > 0 then the state sx is forced to start *)
			state:= LIMIT(0,SX,3);
			last := tx;
			(* this is to avoid to reset sx from the calling programm it does work fine on codesys but i am not sure about other systems, because we are writing to an input *)
			SL := FALSE;
		ELSE
			CASE state OF
				0 :	(* wait for T0 and switch to next cycle *)
					IF tx - last >= T0 THEN
						state := 1;
						last := tx;
					END_IF;
				1 : (* wait for T1 over 1st cycle *)
					IF tx - last >= T1 THEN
						state := 2;
						last := tx;
					END_IF;
				2 : (* wait for T1 over 1st cycle *)
					IF tx - last >= T2 THEN
						state := 3;
						last := tx;
					END_IF;
				3 : (* wait for T2 over 2nd cycle *)
					IF tx - last >= T3 THEN
						IF S0 THEN State := 0; END_IF; (* if S0 is false, the sequence stops at state 3 *)
						last := tx;
					END_IF;
			END_CASE;
		END_IF;
	ELSE
		state := 0;
		last := tx;
	END_IF;

END_FUNCTION_BLOCK

PROGRAM program0
  VAR
	E  :	BOOL ;
	T0 :	TIME;
	T1 :	TIME;
	T2 :	TIME;
	T3 :	TIME;
	S0 :	BOOL;
	SX :	INT;
	SL :	BOOL;

	STATE :	INT;

	func_block : CYCLE_4;
  END_VAR
	func_block.E   :=E ;
	func_block.T0  :=T0;
	func_block.T1  :=T1;
	func_block.T2  :=T2;
	func_block.T3  :=T3;
	func_block.S0  :=S0;
	func_block.SX  :=SX;
	func_block.SL  :=SL;
	func_block();
	STATE := func_block.STATE;
END_PROGRAM

CONFIGURATION Config0
	VAR_GLOBAL
		PLC_TICKS_PER_SEC :	INT;
		PLC_SYS_TICK_CNT :	DINT;
	END_VAR

  	RESOURCE Res0 ON PLC
    	TASK task0(INTERVAL := T#20ms,PRIORITY := 0);
    	PROGRAM instance0 WITH task0 : program0;
  	END_RESOURCE
END_CONFIGURATION

(* ---- CYCLE_TIME.ST ---- *)
FUNCTION_BLOCK T_PLC_MS_block
	VAR_OUTPUT
		T_PLC_MS :	UDINT;
	END_VAR

	VAR_EXTERNAL
		PLC_TICKS_PER_SEC :	INT;
		PLC_SYS_TICK_CNT :	DINT;
	END_VAR

	VAR
		debug :	BOOL;(*Debug-Mode ON / OFF*)
		N :	INT;(*Debug-Faktor*)
		Offset :	UDINT;(*Debug-Offset*)
		temp :	DWORD := DWORD#1;(*Debug-Offset*)
		mode :	BOOL;(*modus*)
		faktor :	UDINT;(*Systemtakt-Faktor*)
		init :	BOOL;
		v_plc_ticks_per_sec :	UDINT;
		base :	UDINT := UDINT#1000;
	END_VAR

	IF init = FALSE THEN
		v_plc_ticks_per_sec := INT_TO_UDINT(PLC_TICKS_PER_SEC);
		IF v_plc_ticks_per_sec = UDINT#1024 THEN
			faktor := UDINT#1;
			mode := FALSE;
		ELSIF v_plc_ticks_per_sec > UDINT#0 THEN
			IF v_plc_ticks_per_sec <= base THEN
				faktor := base / v_plc_ticks_per_sec;
				mode := FALSE;
			ELSE
				faktor := v_plc_ticks_per_sec / base;
				mode := TRUE;
			END_IF;
		ELSE
			faktor := UDINT#1;
		END_IF;
		init := TRUE;
	END_IF;

	IF mode THEN
		T_PLC_MS := DINT_TO_UDINT(PLC_SYS_TICK_CNT) / faktor;
	ELSE
		T_PLC_MS := DINT_TO_UDINT(PLC_SYS_TICK_CNT) * faktor;
	END_IF;

	IF debug THEN
		T_PLC_MS := (DWORD_TO_UDINT(SHL(UDINT_TO_DWORD(T_PLC_MS),N) OR SHL(temp,N)) - UDINT#1) + Offset;
	END_IF;

END_FUNCTION_BLOCK

FUNCTION_BLOCK CYCLE_TIME
	VAR_INPUT
		RST :	BOOL;
	END_VAR

	VAR_OUTPUT
		CT_MIN :	TIME := t#0s;
		CT_MAX :	TIME := t#0s;
		CT_LAST :	TIME;
		SYSTIME :	TIME;
		SYSDAYS :	INT;
		CYCLES :	DWORD;
	END_VAR

	VAR
		last_cycle :	TIME;
		tx :	TIME;
		init :	BOOL;
		T_PLC_MS :	T_PLC_MS_block;
	END_VAR

	T_PLC_MS();
	tx:= UDINT_TO_TIME(T_PLC_MS.T_PLC_MS) - last_cycle;

	IF rst THEN
		ct_min := t#10h;
		ct_max := t#0ms;
		cycles := DWORD#0;
	ELSIF last_cycle > t#0s THEN
		IF tx < ct_min THEN ct_min := tx;
		ELSIF tx > ct_max THEN ct_max := tx;
		END_IF;
		ct_last := tx;
	ELSIF ct_min = t#0s THEN
		ct_min := t#0s - t#1ms;
	END_IF;
	IF init THEN
		systime := systime + tx;
			IF systime >= t#1d THEN
				systime := systime - t#1d;
				sysdays := sysdays + 1;
			END_IF;
	END_IF;
	init := TRUE;
	last_cycle := last_cycle + tx;
	cycles := UDINT_TO_DWORD(DWORD_TO_UDINT(cycles) + UDINT#1);

END_FUNCTION_BLOCK

PROGRAM program0
  VAR
	RST :	BOOL;

	CT_MIN  :	TIME;
	CT_MAX  :	TIME;
	CT_LAST :	TIME;
	SYSTIME :	TIME;
	SYSDAYS :	INT;
	CYCLES  :	DWORD;

	func_block : CYCLE_TIME;
  END_VAR
	func_block.RST   :=RST ;
	func_block();
	CT_MIN := func_block.CT_MIN ;
	CT_MAX := func_block.CT_MAX ;
	CT_LAST:= func_block.CT_LAST;
	SYSTIME:= func_block.SYSTIME;
	SYSDAYS:= func_block.SYSDAYS;
	CYCLES := func_block.CYCLES ;
END_PROGRAM

CONFIGURATION Config0
	VAR_GLOBAL
		PLC_TICKS_PER_SEC :	INT;
		PLC_SYS_TICK_CNT :	DINT;
	END_VAR

  	RESOURCE Res0 ON PLC
    	TASK task0(INTERVAL := T#20ms,PRIORITY := 0);
    	PROGRAM instance0 WITH task0 : program0;
  	END_RESOURCE
END_CONFIGURATION

(* ---- D_TRIG.ST ---- *)
FUNCTION_BLOCK D_TRIG
	VAR_INPUT
		IN :	DWORD;
	END_VAR

	VAR_OUTPUT
		Q :	BOOL;
		X :	DWORD;
	END_VAR

	VAR
		last_in :	DWORD;
	END_VAR

	Q := in <> last_in;
	X := UDINT_TO_DWORD(DWORD_TO_UDINT(in) - DWORD_TO_UDINT(last_in));
	last_in := in;
END_FUNCTION_BLOCK

PROGRAM program0
  VAR
	IN :	DWORD;

	Q :	BOOL;
	X :	DWORD;

	func_block : D_TRIG;
  END_VAR
	func_block.IN  := IN;
	func_block();
	Q := func_block.Q;
	X := func_block.X;
END_PROGRAM

CONFIGURATION Config0
  RESOURCE Res0 ON PLC
    TASK task0(INTERVAL := T#20ms,PRIORITY := 0);
    PROGRAM instance0 WITH task0 : program0;
  END_RESOURCE
END_CONFIGURATION

(* ---- DATE_TO_STRING.ST ---- *)
FUNCTION YEAR_OF_DATE:INT
	VAR_INPUT
		IDATE :	UDINT;
	END_VAR

	YEAR_OF_DATE := UDINT_TO_INT((idate+UDINT#43200) / UDINT#31557600 + UDINT#1970);
END_FUNCTION

FUNCTION DAY_OF_YEAR:INT
	VAR_INPUT
		IDATE :	UDINT;
	END_VAR

	DAY_OF_YEAR := UDINT_TO_INT(((idate) / UDINT#86400) MOD UDINT#1461);
	IF DAY_OF_YEAR > 729 THEN
		IF DAY_OF_YEAR > 1095 THEN DAY_OF_YEAR := DAY_OF_YEAR - 1095; ELSE DAY_OF_YEAR := DAY_OF_YEAR - 729; END_IF;
	ELSIF DAY_OF_YEAR > 364 THEN
		DAY_OF_YEAR := DAY_OF_YEAR - 364;
	ELSE
		DAY_OF_YEAR := DAY_OF_YEAR + 1;
	END_IF;
END_FUNCTION

FUNCTION LEAP_OF_DATE:BOOL

	VAR_INPUT
		IDATE :	UDINT;
	END_VAR

	LEAP_OF_DATE := SHL(UDINT_TO_DWORD((idate + UDINT#43200) / UDINT#31557600), 30) = DWORD#16#80000000;
END_FUNCTION

FUNCTION MONTH_OF_DATE:INT

	VAR_INPUT
		IDATE :	UDINT;
	END_VAR

	MONTH_OF_DATE := DAY_OF_YEAR(idate);
	IF MONTH_OF_DATE < 32 THEN
		MONTH_OF_DATE := 1;
	ELSIF LEAP_OF_DATE((IDATE)) THEN
		MONTH_OF_DATE := (MONTH_OF_DATE * 53 + 1668) / 1623;
	ELSE
		MONTH_OF_DATE := (MONTH_OF_DATE * 53 + 1700) / 1620;
	END_IF;
END_FUNCTION

FUNCTION DAY_OF_MONTH:INT
	VAR_INPUT
		IDATE :	UDINT;
	END_VAR

	day_of_month := day_of_year(idate);

	IF leap_of_Date((idate)) THEN
		CASE day_of_month OF
			32..60	:	day_of_month := day_of_month - 31;
			61..91	:	day_of_month := day_of_month - 60;
			92..121 :	day_of_month := day_of_month - 91;
			122..152:	day_of_month := day_of_month - 121;
			153..182:	day_of_month := day_of_month - 152;
			183..213:	day_of_month := day_of_month - 182;
			214..244:	day_of_month := day_of_month - 213;
			245..274:	day_of_month := day_of_month - 244;
			275..305:	day_of_month := day_of_month - 274;
			306..335:	day_of_month := day_of_month - 305;
			336..366:	day_of_month := day_of_month - 335;
		END_CASE;
	ELSE
		CASE day_of_month OF
			32..59	:	day_of_month := day_of_month - 31;
			60..90	:	day_of_month := day_of_month - 59;
			91..120 :	day_of_month := day_of_month - 90;
			121..151:	day_of_month := day_of_month - 120;
			152..181:	day_of_month := day_of_month - 151;
			182..212:	day_of_month := day_of_month - 181;
			213..243:	day_of_month := day_of_month - 212;
			244..273:	day_of_month := day_of_month - 243;
			274..304:	day_of_month := day_of_month - 273;
			305..334:	day_of_month := day_of_month - 304;
			335..365:	day_of_month := day_of_month - 334;
		END_CASE;
	END_IF;
END_FUNCTION

FUNCTION_BLOCK DATE_TO_STRING2
	VAR_INPUT
		IDATE :	UDINT;
	END_VAR

	VAR_OUTPUT
		DATE_STRING :	STRING;
	END_VAR

	VAR
		st_tmp1 :	STRING;
	END_VAR

	st_tmp1 := CONCAT(INT_TO_STRING(YEAR_OF_DATE(IDATE)),INT_TO_STRING(MONTH_OF_DATE(IDATE)));
	DATE_STRING := CONCAT(st_tmp1,INT_TO_STRING(day_of_month(IDATE)));
END_FUNCTION_BLOCK

PROGRAM program0
  VAR
    LocalVar0 : UDINT;
	LocalOUT  : STRING;
	func_block : DATE_TO_STRING2;
  END_VAR
	func_block.IDATE  := LocalVar0;
	func_block();
	LocalOUT := func_block.DATE_STRING;
END_PROGRAM

CONFIGURATION Config0
  RESOURCE Res0 ON PLC
    TASK task0(INTERVAL := T#20ms,PRIORITY := 0);
    PROGRAM instance0 WITH task0 : program0;
  END_RESOURCE
END_CONFIGURATION

(* ---- DEAD_BAND_A.ST ---- *)
FUNCTION_BLOCK T_PLC_US_Block

	VAR_OUTPUT
		T_PLC_US :	UDINT;
	END_VAR

	VAR_EXTERNAL
		PLC_TICKS_PER_SEC :	INT;
		PLC_SYS_TICK_CNT :	DINT;
	END_VAR

	VAR
		debug :	BOOL;
		N :	INT;
		Offset :	UDINT;
		temp :	DWORD := DWORD#1;
		mode :	BOOL;
		faktor :	UDINT;
		init :	BOOL;
		v_plc_ticks_per_sec :	UDINT;
		base :	UDINT := UDINT#1000000;
	END_VAR

	IF init = FALSE THEN
		v_plc_ticks_per_sec := INT_TO_UDINT(PLC_TICKS_PER_SEC);
		IF v_plc_ticks_per_sec = UDINT#1024 THEN
			faktor := UDINT#1000;
			mode := FALSE;
		ELSIF v_plc_ticks_per_sec > UDINT#0 THEN
			IF v_plc_ticks_per_sec <= base THEN
				faktor := base / v_plc_ticks_per_sec;
				mode := FALSE;
			ELSE
				faktor := v_plc_ticks_per_sec / base;
				mode := TRUE;
			END_IF;
		ELSE
			faktor := UDINT#1;
		END_IF;
		init := TRUE;
	END_IF;

	IF mode THEN
		T_PLC_US := DINT_TO_UDINT(PLC_SYS_TICK_CNT) / faktor;
	ELSE
		T_PLC_US := DINT_TO_UDINT(PLC_SYS_TICK_CNT) * faktor;
	END_IF;

	IF debug THEN
		T_PLC_US := (DWORD_TO_UDINT(SHL(UDINT_TO_DWORD(T_PLC_US),N) OR SHL(temp,N)) - UDINT#1) + Offset;
	END_IF;
END_FUNCTION_BLOCK

FUNCTION_BLOCK FT_PT1

	VAR_INPUT
		IN :	REAL;
		T :	TIME;
		K :	REAL := 1.0;
	END_VAR

	VAR_OUTPUT
		OUT :	REAL;
	END_VAR

	VAR
		last :	UDINT;
		tx :	UDINT;
		init :	BOOL;
		T_PLC_US :	T_PLC_US_Block;
	END_VAR

	T_PLC_US();
	tx:= T_PLC_US.T_PLC_US;

	IF NOT init OR T = t#0s THEN
		init := TRUE;
		out := K * in;
	ELSE
		out := out + (in * K - out) * UDINT_TO_REAL(Tx - last) / TIME_TO_REAL(T) * 1.0E-3;
		IF ABS(out) < 1.0E-20 THEN out := 0.0; END_IF;
	END_IF;
	last := tx;
END_FUNCTION_BLOCK

FUNCTION _REAL_TO_DWORD: DWORD

  VAR_INPUT
    X :	REAL;
  END_VAR

  IF REAL_TO_DWORD(0.5) = DWORD#1 THEN
    _REAL_TO_DWORD := REAL_TO_DWORD(x);
  ELSIF X > 0.0 THEN
    _REAL_TO_DWORD := REAL_TO_DWORD(x+0.5);
  ELSIF X < 0.0 THEN
    _REAL_TO_DWORD := REAL_TO_DWORD(x-0.5);
  ELSE
    _REAL_TO_DWORD := DWORD#0;
  END_IF;
END_FUNCTION

FUNCTION _DWORD_TO_REAL:REAL
	VAR_INPUT
		IN :	DWORD;
	END_VAR

	_DWORD_TO_REAL := UDINT_TO_REAL(DWORD_TO_UDINT(IN));
END_FUNCTION

FUNCTION MULTIME:TIME
	VAR_INPUT
		T :	TIME;
		M :	REAL;
	END_VAR

	multime := DWORD_TO_TIME(_REAL_TO_DWORD(_DWORD_TO_REAL(TIME_TO_DWORD(t))*M));
END_FUNCTION

FUNCTION_BLOCK DEAD_BAND_A
	VAR_INPUT
		X :	REAL;
		T :	TIME;
		KL :	REAL := 1.0;
		LM :	REAL;
	END_VAR

	VAR_OUTPUT
		Y :	REAL;
		L :	REAL;
	END_VAR

	VAR
		tp1 :	FT_PT1;
		tp2 :	FT_PT1;
	END_VAR

	tp1(in := X, T:= T);
	tp2(in := ABS(tp1.out - X), T := MULTIME(T, 4.0));
	L := MIN(KL * tp2.out, LM);

	IF X > L THEN
		Y := X - L;
	ELSIF X < -L THEN
		Y := X + L;
	ELSE
		Y := 0.0;
	END_IF;
END_FUNCTION_BLOCK

PROGRAM program0
  VAR

		X  :	REAL;
		T  :	TIME;
		KL :	REAL;
		LM :	REAL;

		Y :	REAL;
		L :	REAL;

	func_block : DEAD_BAND_A;
  END_VAR
	func_block.X   :=X ;
	func_block.T   :=T ;
	func_block.KL  :=KL;
	func_block.LM  :=LM;
	func_block();
	Y := func_block.Y;
	L := func_block.L;
END_PROGRAM

CONFIGURATION Config0

	VAR_GLOBAL
		PLC_TICKS_PER_SEC :	INT;
		PLC_SYS_TICK_CNT :	DINT;
	END_VAR

	RESOURCE Res0 ON PLC
		TASK task0(INTERVAL := T#20ms,PRIORITY := 0);
		PROGRAM instance0 WITH task0 : program0;
	END_RESOURCE

END_CONFIGURATION

(* ---- DEAD_ZONE2.ST ---- *)
FUNCTION_BLOCK DEAD_ZONE2
	VAR_INPUT
		X :	REAL;
		L :	REAL;
	END_VAR

	VAR_OUTPUT
		Y :	REAL;
	END_VAR

	IF ABS(x) > L THEN
		Y := X;
	ELSIF Y > 0.0 THEN
		Y := L;
	ELSE
		Y := -L;
	END_IF;
END_FUNCTION_BLOCK

PROGRAM program0
  VAR
    LocalVar0 : REAL;
	LocalVar1 : REAL;
	LocalOUT  : REAL;
	func_block : DEAD_ZONE2;
  END_VAR
	func_block.X  := LocalVar0;
	func_block.L  := LocalVar1;
	func_block();
	LocalOUT := func_block.Y;
END_PROGRAM

CONFIGURATION Config0
  RESOURCE Res0 ON PLC
    TASK task0(INTERVAL := T#20ms,PRIORITY := 0);
    PROGRAM instance0 WITH task0 : program0;
  END_RESOURCE
END_CONFIGURATION

(* ---- DEBOUNCE.ST ---- *)
FUNCTION_BLOCK DEBOUNCE_Block

	VAR_INPUT
		IN :	BOOL;
		TD :	TIME;
		PM :	BOOL;
	END_VAR

	VAR_OUTPUT
		Q :	BOOL;
	END_VAR

	VAR
		deb :	TOF;
	END_VAR

	IF NOT deb.Q AND IN THEN
		Q := TRUE;
	ELSIF NOT PM THEN
		Q := deb.Q;
	ELSE
		Q := FALSE;
	END_IF;

END_FUNCTION_BLOCK

PROGRAM program0
	VAR
		IN :	BOOL;
		TD :	TIME;
		PM :	BOOL;
		Q :	BOOL;

		func_block : DEBOUNCE_Block;
	END_VAR
	func_block.IN := IN;
	func_block.TD := TD;
	func_block.PM := PM ;

	func_block();
	Q  := func_block.Q;
END_PROGRAM

CONFIGURATION Config0
	RESOURCE Res0 ON PLC
		TASK task0(INTERVAL := T#20ms,PRIORITY := 0);
		PROGRAM instance0 WITH task0 : program0;
	END_RESOURCE
END_CONFIGURATION

(* ---- DEC_2.ST ---- *)
FUNCTION_BLOCK DEC_2
	VAR_INPUT
		D :	BOOL;
		A :	BOOL;
	END_VAR
	VAR_OUTPUT
		Q0 :	BOOL;
		Q1 :	BOOL;
	END_VAR
	Q0 := D AND NOT A;
	Q1 := D AND A;
END_FUNCTION_BLOCK

PROGRAM program0
  VAR
    LocalVar0 : BOOL;
	LocalVar1 : BOOL;
	LocalOUT  : BOOL;
	LocalOUT1  : BOOL;
	func_block : DEC_2;
  END_VAR
	func_block.D  := LocalVar0;
	func_block.A  := LocalVar1;
	func_block();
	LocalOUT := func_block.Q0;
	LocalOUT1 := func_block.Q1;
END_PROGRAM

CONFIGURATION Config0
  RESOURCE Res0 ON PLC
    TASK task0(INTERVAL := T#20ms,PRIORITY := 0);
    PROGRAM instance0 WITH task0 : program0;
  END_RESOURCE
END_CONFIGURATION

(* ---- DEC_4.ST ---- *)
FUNCTION_BLOCK DEC_4
	VAR_INPUT
		D :	BOOL;
		A0 :	BOOL;
		A1 :	BOOL;
	END_VAR

	VAR_OUTPUT
		Q0 :	BOOL;
		Q1 :	BOOL;
		Q2 :	BOOL;
		Q3 :	BOOL;
	END_VAR

	Q0 := D AND NOT A0 AND NOT A1;
	Q1 := D AND A0 AND NOT A1;
	Q2 := D AND NOT A0 AND A1;
	Q3 := D AND A0 AND A1;
END_FUNCTION_BLOCK

PROGRAM program0
  VAR
	D :	BOOL;
	A0 :	BOOL;
	A1 :	BOOL;

	Q0 :	BOOL;
	Q1 :	BOOL;
	Q2 :	BOOL;
	Q3 :	BOOL;

	func_block : DEC_4;
  END_VAR
	func_block.D   := D  ;
	func_block.A0  := A0  ;
	func_block.A1  := A1  ;
	func_block();
	Q0:= func_block.Q0;
	Q1:= func_block.Q1;
	Q2:= func_block.Q2;
	Q3:= func_block.Q3;
END_PROGRAM

CONFIGURATION Config0
  RESOURCE Res0 ON PLC
    TASK task0(INTERVAL := T#20ms,PRIORITY := 0);
    PROGRAM instance0 WITH task0 : program0;
  END_RESOURCE
END_CONFIGURATION

(* ---- DEC_8.ST ---- *)
FUNCTION BIT_LOAD_B:BYTE
	VAR_INPUT
		IN :	BYTE;
		VAL :	BOOL;
		POS :	INT;
	END_VAR

	IF VAL THEN
		BIT_LOAD_B := in OR SHL(BYTE#1,pos);
	ELSE
		BIT_LOAD_B := in AND (NOT SHL(BYTE#1,pos));
	END_IF;
END_FUNCTION

FUNCTION _BYTE_TO_INT:INT
	VAR_INPUT
		IN :	BYTE;
	END_VAR

	_BYTE_TO_INT := USINT_TO_INT(BYTE_TO_USINT(IN));
END_FUNCTION

FUNCTION_BLOCK DEC_8

	VAR_INPUT
		D :	BOOL;
		A0 :	BOOL;
		A1 :	BOOL;
		A2 :	BOOL;
	END_VAR

	VAR_OUTPUT
		Q0 :	BOOL;
		Q1 :	BOOL;
		Q2 :	BOOL;
		Q3 :	BOOL;
		Q4 :	BOOL;
		Q5 :	BOOL;
		Q6 :	BOOL;
		Q7 :	BOOL;
	END_VAR

	VAR
		X :	BYTE;
	END_VAR

	X:=BIT_LOAD_B(X,A0,0); (* X.0 := A0; *)
	X:=BIT_LOAD_B(X,A1,1); (* X.1 := A1; *)
	X:=BIT_LOAD_B(X,A2,2); (* X.2 := A2; *)

	Q0 := FALSE;
	Q1 := FALSE;
	Q2 := FALSE;
	Q3 := FALSE;
	Q4 := FALSE;
	Q5 := FALSE;
	Q6 := FALSE;
	Q7 := FALSE;

	CASE _BYTE_TO_INT(X) OF
		0 : Q0 := D;
		1 : Q1 := D;
		2 : Q2 := D;
		3 : Q3 := D;
		4 : Q4 := D;
		5 : Q5 := D;
		6 : Q6 := D;
		7 : Q7 := D;
	END_CASE;

	END_FUNCTION_BLOCK

PROGRAM program0
  VAR
	D :	BOOL;
	A0 :	BOOL;
	A1 :	BOOL;
	A2 :	BOOL;

	Q0 :	BOOL;
	Q1 :	BOOL;
	Q2 :	BOOL;
	Q3 :	BOOL;
	Q4 :	BOOL;
	Q5 :	BOOL;
	Q6 :	BOOL;
	Q7 :	BOOL;

	func_block : DEC_8;
  END_VAR
	func_block.D   := D  ;
	func_block.A0  := A0  ;
	func_block.A1  := A1  ;
	func_block.A2  := A2  ;
	func_block();
	Q0:= func_block.Q0;
	Q1:= func_block.Q1;
	Q2:= func_block.Q2;
	Q3:= func_block.Q3;
	Q4:= func_block.Q4;
	Q5:= func_block.Q5;
	Q6:= func_block.Q6;
	Q7:= func_block.Q7;
END_PROGRAM

CONFIGURATION Config0
  RESOURCE Res0 ON PLC
    TASK task0(INTERVAL := T#20ms,PRIORITY := 0);
    PROGRAM instance0 WITH task0 : program0;
  END_RESOURCE
END_CONFIGURATION

(* ---- DEG_TO_DIR.ST ---- *)
TYPE oscat_LANGUAGE:
  STRUCT
    DEFAULT 	: INT;
	LMAX    	: INT;
  END_STRUCT;
END_TYPE

TYPE
  oscat_ELEMENT_DIRS 		: ARRAY [0..15] OF STRING;
  oscat_DIRS				: ARRAY [1..3]  OF oscat_ELEMENT_DIRS := [0,0 , 0];
END_TYPE

FUNCTION_BLOCK SETUP_DIRS
	VAR_IN_OUT
		DIRS :	oscat_DIRS;
	END_VAR

	VAR
		init :	BOOL;
	END_VAR

	IF init THEN RETURN; END_IF;
	init := TRUE;

	(* ---- english --- *)
	DIRS[1][00] := 'N';
	DIRS[1][01] := 'NNE';
	DIRS[1][02] := 'NE';
	DIRS[1][03] := 'ENE';
	DIRS[1][04] := 'E';
	DIRS[1][05] := 'ESE';
	DIRS[1][06] := 'SE';
	DIRS[1][07] := 'SSE';
	DIRS[1][08] := 'S';
	DIRS[1][09] := 'SSW';
	DIRS[1][10] := 'SW';
	DIRS[1][11] := 'WSW';
	DIRS[1][12] := 'W';
	DIRS[1][13] := 'WNW';
	DIRS[1][14] := 'NW';
	DIRS[1][15] := 'NNW';

	(* ---- german --- *)
	DIRS[2][00] := 'N';
	DIRS[2][01] := 'NNO';
	DIRS[2][02] := 'NO';
	DIRS[2][03] := 'ONO';
	DIRS[2][04] := 'O';
	DIRS[2][05] := 'OSO';
	DIRS[2][06] := 'SO';
	DIRS[2][07] := 'SSO';
	DIRS[2][08] := 'S';
	DIRS[2][09] := 'SSW';
	DIRS[2][10] := 'SW';
	DIRS[2][11] := 'WSW';
	DIRS[2][12] := 'W';
	DIRS[2][13] := 'WNW';
	DIRS[2][14] := 'NW';
	DIRS[2][15] := 'NNW';

	(* ---- french --- *)
	DIRS[3][00] := 'N';
	DIRS[3][01] := 'NNO';
	DIRS[3][02] := 'NO';
	DIRS[3][03] := 'ONO';
	DIRS[3][04] := 'O';
	DIRS[3][05] := 'OSO';
	DIRS[3][06] := 'SO';
	DIRS[3][07] := 'SSO';
	DIRS[3][08] := 'S';
	DIRS[3][09] := 'SSW';
	DIRS[3][10] := 'SW';
	DIRS[3][11] := 'WSW';
	DIRS[3][12] := 'W';
	DIRS[3][13] := 'WNW';
	DIRS[3][14] := 'NW';
	DIRS[3][15] := 'NNW';
END_FUNCTION_BLOCK

FUNCTION_BLOCK SETUP_LANGUAGE_Block

	VAR_IN_OUT
		LANGUAGE :	oscat_LANGUAGE;
	END_VAR

	VAR
		init :	BOOL;
	END_VAR

	IF init THEN RETURN; END_IF;
	init := TRUE;

	LANGUAGE.DEFAULT  := 1; (* 1=english, 2=german 3=french *)
	LANGUAGE.LMAX := 3;

END_FUNCTION_BLOCK

FUNCTION_BLOCK DEG_TO_DIR_Block
	VAR_INPUT
		DEG :	INT;
		N :	INT;
		L :	INT;
	END_VAR

	VAR_OUTPUT
		DEG_TO_DIR :	STRING;
	END_VAR

	VAR
		ly :	INT;
		y :	INT;
		SETUP_DIRSS :	SETUP_DIRS;
		DIRS :	oscat_DIRS;
		SETUP_LANGUAGE :	SETUP_LANGUAGE_Block;
		LANGUAGE :	oscat_LANGUAGE;
	END_VAR

	SETUP_DIRSS(DIRS:=DIRS);
	DIRS:=SETUP_DIRSS.DIRS;
	SETUP_LANGUAGE(LANGUAGE:=LANGUAGE);
	LANGUAGE:=SETUP_LANGUAGE.LANGUAGE;

	IF L = 0 THEN ly := LANGUAGE.DEFAULT; ELSE ly := MIN(L, LANGUAGE.LMAX); END_IF;
	y := ((WORD_TO_INT(SHL(INT_TO_WORD(DEG),N-1)) + 45) / 90) MOD WORD_TO_INT(SHL(WORD#2,N))* WORD_TO_INT(SHR(WORD#8,N));
	DEG_TO_DIR := DIRS[ly][y];
END_FUNCTION_BLOCK

PROGRAM program0

	VAR
		DEG :	INT;
		N   :	INT;
		L   :	INT;

		DEG_TO_DIR :	STRING;

		func_block : DEG_TO_DIR_Block;
	END_VAR
		func_block.DEG:=DEG;
		func_block.N  :=N  ;
		func_block.L  :=L  ;

		func_block();
		DEG_TO_DIR := func_block.DEG_TO_DIR;

END_PROGRAM

CONFIGURATION Config0

	RESOURCE Res0 ON PLC
		TASK task0(INTERVAL := T#20ms,PRIORITY := 0);
		PROGRAM instance0 WITH task0 : program0;
	END_RESOURCE

END_CONFIGURATION

(* ---- DEL_CHARS.ST ---- *)
FUNCTION_BLOCK DEL_CHARS_Block
	VAR_INPUT
		IN :	STRING;
		CX :	STRING;
	END_VAR

	VAR_OUTPUT
		DEL_CHARS :	STRING;
	END_VAR

	VAR
		pos :	INT;
		stop :	INT;
		char :	STRING;
	END_VAR

	DEL_CHARS := IN;
	stop := LEN(in);
	pos := 1;
	WHILE pos <= stop DO
		char := MID(DEL_CHARS, 1, pos);
		IF FIND(cx,char) > 0 THEN
			DEL_CHARS := DELETE(DEL_CHARS, 1, pos);
			stop := stop - 1;
		ELSE
			pos := pos + 1;
		END_IF;
	END_WHILE;

END_FUNCTION_BLOCK

PROGRAM program0
  VAR
    LocalVar0 : STRING;
	LocalVar1 : STRING;
	LocalOUT  : STRING;
	func_block : DEL_CHARS_Block;
  END_VAR
	func_block.IN := LocalVar0;
	func_block.CX  := LocalVar1;
	func_block();
	LocalOUT := func_block.DEL_CHARS;
END_PROGRAM

CONFIGURATION Config0
  RESOURCE Res0 ON PLC
    TASK task0(INTERVAL := T#20ms,PRIORITY := 0);
    PROGRAM instance0 WITH task0 : program0;
  END_RESOURCE
END_CONFIGURATION

(* ---- DELAY.ST ---- *)
TYPE
	oscat_delay_buf             : ARRAY [0..31]   OF REAL;
END_TYPE

FUNCTION INC1:INT

	VAR_INPUT
		X :	INT;
		N :	INT;
	END_VAR

	IF X >= N - 1 THEN
		INC1 := 0;
	ELSE
		INC1 := X + 1;
	END_IF;
END_FUNCTION

FUNCTION_BLOCK DELAY

	VAR_INPUT
		IN :	REAL;
		N :	INT;
		RST :	BOOL;
	END_VAR

	VAR_OUTPUT
		OUT :	REAL;
	END_VAR

	VAR
		buf :	oscat_delay_buf;
		i :	INT;
		init :	BOOL;
		stop :	INT;
	END_VAR

	stop := LIMIT(0,N,32) - 1;
	IF rst OR NOT init THEN
		init := TRUE;
		FOR i := 0 TO stop DO buf[i] := in; END_FOR;
		out := in;
		i := 0;
	ELSIF stop < 0 THEN
		out := in;
	ELSE
		out := buf[i];
		buf[i] := in;
		i := INC1(i, N);
	END_IF;

END_FUNCTION_BLOCK

PROGRAM program0
  VAR
	IN :	REAL;
	N :	INT;
	RST :	BOOL;
	OUT :	REAL;
	func_block : DELAY;
  END_VAR
	func_block.IN  :=IN;
	func_block.N  :=N;
	func_block.RST  :=RST;
	func_block();
	OUT := func_block.OUT;

END_PROGRAM

CONFIGURATION Config0
	RESOURCE Res0 ON PLC
		TASK task0(INTERVAL := T#20ms,PRIORITY := 0);
		PROGRAM instance0 WITH task0 : program0;
	END_RESOURCE
END_CONFIGURATION

(* ---- DELAY_4.ST ---- *)
FUNCTION_BLOCK DELAY_4

	VAR_INPUT
		IN :	REAL;
	END_VAR

	VAR_OUTPUT
		OUT1 :	REAL;
		OUT2 :	REAL;
		OUT3 :	REAL;
		OUT4 :	REAL;
	END_VAR

	VAR
		temp :	REAL;
	END_VAR

	out4 := out3;
	out3 := out2;
	out2 := out1;
	out1 := temp;
	temp := in;

END_FUNCTION_BLOCK

PROGRAM program0
  VAR
	IN :	REAL;

	OUT1 :	REAL;
	OUT2 :	REAL;
	OUT3 :	REAL;
	OUT4 :	REAL;
	func_block : DELAY_4;
  END_VAR
	func_block.IN  := IN;
	func_block();
	OUT1:= func_block.OUT1;
	OUT2:= func_block.OUT2;
	OUT3:= func_block.OUT3;
	OUT4:= func_block.OUT4;
END_PROGRAM

CONFIGURATION Config0
  RESOURCE Res0 ON PLC
    TASK task0(INTERVAL := T#20ms,PRIORITY := 0);
    PROGRAM instance0 WITH task0 : program0;
  END_RESOURCE
END_CONFIGURATION

(* ---- DIMM_2.ST ---- *)
FUNCTION UDINT_TO_TIME2:TIME

	VAR_INPUT
		IN :	UDINT;
	END_VAR

	UDINT_TO_TIME2 := DINT_TO_TIME(UDINT_TO_DINT(IN));

END_FUNCTION

FUNCTION_BLOCK T_PLC_MS_block
	VAR_OUTPUT
		T_PLC_MS :	UDINT;
	END_VAR

	VAR_EXTERNAL
		PLC_TICKS_PER_SEC :	INT;
		PLC_SYS_TICK_CNT :	DINT;
	END_VAR

	VAR
		debug :	BOOL;(*Debug-Mode ON / OFF*)
		N :	INT;(*Debug-Faktor*)
		Offset :	UDINT;(*Debug-Offset*)
		temp :	DWORD := DWORD#1;(*Debug-Offset*)
		mode :	BOOL;(*modus*)
		faktor :	UDINT;(*Systemtakt-Faktor*)
		init :	BOOL;
		v_plc_ticks_per_sec :	UDINT;
		base :	UDINT := UDINT#1000;
	END_VAR

	IF init = FALSE THEN
		v_plc_ticks_per_sec := INT_TO_UDINT(PLC_TICKS_PER_SEC);
		IF v_plc_ticks_per_sec = UDINT#1024 THEN
			faktor := UDINT#1;
			mode := FALSE;
		ELSIF v_plc_ticks_per_sec > UDINT#0 THEN
			IF v_plc_ticks_per_sec <= base THEN
				faktor := base / v_plc_ticks_per_sec;
				mode := FALSE;
			ELSE
				faktor := v_plc_ticks_per_sec / base;
				mode := TRUE;
			END_IF;
		ELSE
			faktor := UDINT#1;
		END_IF;
		init := TRUE;
	END_IF;

	IF mode THEN
		T_PLC_MS := DINT_TO_UDINT(PLC_SYS_TICK_CNT) / faktor;
	ELSE
		T_PLC_MS := DINT_TO_UDINT(PLC_SYS_TICK_CNT) * faktor;
	END_IF;

	IF debug THEN
		T_PLC_MS := (DWORD_TO_UDINT(SHL(UDINT_TO_DWORD(T_PLC_MS),N) OR SHL(temp,N)) - UDINT#1) + Offset;
	END_IF;

END_FUNCTION_BLOCK

FUNCTION TIME_TO_UDINT2:UDINT
	VAR_INPUT
		X :	TIME;
	END_VAR

	TIME_TO_UDINT2 := DINT_TO_UDINT(TIME_TO_DINT(X));
END_FUNCTION

FUNCTION FRMP_B:BYTE
	VAR_INPUT
		START :	BYTE;
		DIR :	BOOL;
		TD :	TIME;
		TR :	TIME;
	END_VAR

	IF TD < TR THEN
		FRMP_B := MIN(UDINT_TO_BYTE(DWORD_TO_UDINT(SHL(TIME_TO_DWORD(TD), 8)) / TIME_TO_UDINT2(TR)), SEL(DIR, START, USINT_TO_BYTE(USINT#255 - BYTE_TO_USINT(START))));
		IF DIR THEN
			FRMP_B := USINT_TO_BYTE(BYTE_TO_USINT(START) + BYTE_TO_USINT(FRMP_B));
		ELSE
			FRMP_B := USINT_TO_BYTE(BYTE_TO_USINT(START) - BYTE_TO_USINT(FRMP_B));
		END_IF;
	ELSE
		FRMP_B := SEL(DIR, BYTE#0, BYTE#255);
	END_IF;
END_FUNCTION

FUNCTION_BLOCK _RMP_B
	VAR_INPUT
		DIR :	BOOL;
		E :	BOOL := TRUE;
		TR :	TIME;
	END_VAR

	VAR_IN_OUT
		RMP :	BYTE;
	END_VAR

	VAR
		T_PLC_MS :	T_PLC_MS_Block;
		tx :	TIME;
		tl :	TIME;
		tn :	TIME;
		init :	BOOL;
		last_dir :	BOOL;
		start :	BYTE;
	END_VAR

	T_PLC_MS();
	tx := UDINT_TO_TIME(T_PLC_MS.T_PLC_MS);

	IF E AND init AND (dir = last_dir) AND (RMP <> SEL(DIR, BYTE#0, BYTE#255)) AND TR = tn THEN
		RMP := FRMP_B(start, DIR, tx - tl, TR);
	ELSE
		init := TRUE;
		tl := tx;
		tn := tr;
		start := RMP;
	END_IF;
	last_dir := dir;
END_FUNCTION_BLOCK

FUNCTION_BLOCK CLICK_MODE_Block

	VAR_INPUT
		IN :	BOOL;
		T_LONG :	TIME := T#500ms;
	END_VAR

	VAR_OUTPUT
		SINGLE :	BOOL;
		DOUBLE :	BOOL;
		LONG :	BOOL;
		TP_LONG :	BOOL;
	END_VAR

	VAR
		Timer :	TP;
		cnt :	INT;
		last :	BOOL;
	END_VAR

	timer(in := IN, PT := T_LONG);
	single := FALSE;
	double := FALSE;

	IF timer.Q THEN
		IF NOT in AND last THEN	cnt := cnt + 1; END_IF;
	ELSE
		CASE cnt OF
			1 : single := TRUE;
			2 : double := TRUE;
		END_CASE;
		cnt := 0;
	END_IF;
	last := in;
	TP_LONG := NOT timer.Q AND (NOT LONG) AND IN;
	LONG := NOT timer.Q AND in;

END_FUNCTION_BLOCK

FUNCTION_BLOCK DIMM_2_Block

	VAR_INPUT
		SET :	BOOL;
		VAL :	BYTE := BYTE#255;
		I1 :	BOOL;
		I2 :	BOOL;
		RST :	BOOL;
		T_DEBOUNCE :	TIME := T#10ms;
		T_ON_MAX :	TIME := T#0h;
		T_DIMM_START :	TIME := T#1s;
		T_DIMM :	TIME := T#3s;
		MIN_ON :	BYTE := BYTE#50;
		MAX_ON :	BYTE := BYTE#255;
		RST_OUT :	BOOL;
		SOFT_DIMM :	BOOL := TRUE;
		DBL1_TOG :	BOOL;
		DBL2_TOG :	BOOL;
		DBL1_SET :	BOOL;
		DBL2_SET :	BOOL;
		DBL1_POS :	BYTE;
		DBL2_POS :	BYTE;
	END_VAR

	VAR_OUTPUT
		Q :	BOOL;
		D1 :	BOOL;
		D2 :	BOOL;
	END_VAR

	VAR_IN_OUT
		_OUT :	BYTE;
	END_VAR

	VAR
		t1 :	TOF;
		t2 :	TOF;
		dc1 :	CLICK_MODE_Block;
		dc2 :	CLICK_MODE_Block;
		t3 :	TON;
		dim :	_RMP_B;
	END_VAR

	t1(IN := I1, PT := T_DEBOUNCE);
	t2(IN := I2, PT := T_DEBOUNCE);
	dc1(in := t1.Q, T_LONG := T_DIMM_START);
	dc2(in := t2.Q, T_LONG := T_DIMM_START);

	IF RST THEN
		IF RST_OUT THEN _OUT := BYTE#0; END_IF;
		Q := FALSE;
		D1 := FALSE;
		D2 := FALSE;
	ELSIF set THEN
		_OUT := VAL;
		Q := TRUE;
	ELSIF dc1.SINGLE THEN
		_OUT := LIMIT(MAX(MIN_ON,BYTE#1), _OUT, MAX_ON);
		Q := TRUE;
	ELSIF dc2.SINGLE THEN
		Q := FALSE;
	ELSIF dc1.TP_LONG THEN
		IF NOT Q THEN
			_OUT := SEL(SOFT_DIMM, LIMIT(MAX(MIN_ON,BYTE#1), _OUT, MAX_ON), BYTE#1);
		END_IF;
		Q := TRUE;
		dim.DIR := TRUE;
	ELSIF dc2.TP_LONG THEN
		dim.DIR := FALSE;
	END_IF;

	IF NOT DBL1_TOG THEN D1 := FALSE; END_IF;
	IF dc1.DOUBLE THEN
		IF DBL1_SET THEN
			_OUT := DBL1_POS;
			Q := TRUE;
		ELSE
			D1 := NOT D1;
		END_IF;
	END_IF;
	IF NOT DBL2_TOG THEN D2 := FALSE; END_IF;
	IF dc2.DOUBLE THEN
		IF DBL2_SET THEN
			_OUT := DBL2_POS;
			Q := TRUE;
		ELSE
			D2 := NOT D2;
		END_IF;
	END_IF;

	dim(dir := dc2.LONG, e := dc1.LONG OR dc2.LONG , TR := T_DIMM, rmp := _OUT);
	_OUT := dim.RMP;

	IF _OUT = BYTE#0 THEN Q := FALSE; END_IF;

	IF t_ON_MAX > t#0s THEN
		t3(in := q, pt := T_ON_MAX);
		Q := Q XOR t3.Q;
	END_IF;

END_FUNCTION_BLOCK

PROGRAM program0
	VAR
	    SET :	BOOL;
		VAL :	BYTE := BYTE#255;
		I1 :	BOOL;
		I2 :	BOOL;
		RST :	BOOL;
		T_DEBOUNCE :	TIME := T#10ms;
		T_ON_MAX :	TIME := T#0h;
		T_DIMM_START :	TIME := T#1s;
		T_DIMM :	TIME := T#3s;
		MIN_ON :	BYTE := BYTE#50;
		MAX_ON :	BYTE := BYTE#255;
		RST_OUT :	BOOL;
		SOFT_DIMM :	BOOL := TRUE;
		DBL1_TOG :	BOOL;
		DBL2_TOG :	BOOL;
		DBL1_SET :	BOOL;
		DBL2_SET :	BOOL;
		DBL1_POS :	BYTE;
		DBL2_POS :	BYTE;
		_OUT :	BYTE := BYTE#0;
		Q :	BOOL;
		D1 :	BOOL;
		D2 :	BOOL;

		func_block : DIMM_2_Block;
  	END_VAR
	func_block.SET := SET;
	func_block.VAL := VAL;
	func_block.I1 := I1;
	func_block.I2 := I2;
	func_block.RST := RST;
	func_block.T_DEBOUNCE := T_DEBOUNCE;
	func_block.T_ON_MAX := T_ON_MAX;
	func_block.T_DIMM_START := T_DIMM_START;
	func_block.T_DIMM := T_DIMM;
	func_block.MIN_ON := MIN_ON;
	func_block.MAX_ON := MAX_ON;
	func_block.RST_OUT := RST_OUT;
	func_block.SOFT_DIMM := SOFT_DIMM;
	func_block.DBL1_TOG := DBL1_TOG;
	func_block.DBL2_TOG := DBL2_TOG;
	func_block.DBL1_SET := DBL1_SET;
	func_block.DBL2_SET := DBL2_SET;
	func_block.DBL1_POS := DBL1_POS;
	func_block.DBL2_POS := DBL2_POS;
	func_block._OUT := _OUT;

	func_block();
	_OUT := func_block._OUT;
	Q := func_block.Q;
	D1 := func_block.D1;
	D2 := func_block.D2;
END_PROGRAM

CONFIGURATION Config0
	VAR_GLOBAL
		PLC_TICKS_PER_SEC :	INT;
		PLC_SYS_TICK_CNT :	DINT;
	END_VAR
  	RESOURCE Res0 ON PLC
    	TASK task0(INTERVAL := T#20ms,PRIORITY := 0);
    	PROGRAM instance0 WITH task0 : program0;
  	END_RESOURCE
END_CONFIGURATION

(* ---- DIMM_I.ST ---- *)
FUNCTION_BLOCK SW_RECONFIG_Block

	VAR_INPUT
		IN :	BOOL;
		TD :	TIME;
		TR :	TIME;
	END_VAR

	VAR_OUTPUT
		Q :	BOOL;
	END_VAR

	VAR
		T1 :	TON;
		T2 :	TON;
		INV :	BOOL;
	END_VAR

	t1(in := IN, PT := TD);

	IF tr > t#0s THEN
		Q := t1.Q XOR inv;
		T2(in := Q, pt := TR);
		IF T2.Q THEN INV := NOT INV; END_IF;
	ELSE
		Q := t1.Q;
	END_IF;

END_FUNCTION_BLOCK

FUNCTION_BLOCK CLICK_MODE_Block

	VAR_INPUT
		IN :	BOOL;
		T_LONG :	TIME := T#500ms;
	END_VAR

	VAR_OUTPUT
		SINGLE :	BOOL;
		DOUBLE :	BOOL;
		LONG :	BOOL;
		TP_LONG :	BOOL;
	END_VAR

	VAR
		Timer :	TP;
		cnt :	INT;
		last :	BOOL;
	END_VAR

	timer(in := IN, PT := T_LONG);
	single := FALSE;
	double := FALSE;

	IF timer.Q THEN
		IF NOT in AND last THEN	cnt := cnt + 1; END_IF;
	ELSE
		CASE cnt OF
			1 : single := TRUE;
			2 : double := TRUE;
		END_CASE;
		cnt := 0;
	END_IF;
	last := in;
	TP_LONG := NOT timer.Q AND (NOT LONG) AND IN;
	LONG := NOT timer.Q AND in;

END_FUNCTION_BLOCK

FUNCTION UDINT_TO_TIME2:TIME

	VAR_INPUT
		IN :	UDINT;
	END_VAR

	UDINT_TO_TIME2 := DINT_TO_TIME(UDINT_TO_DINT(IN));

END_FUNCTION

FUNCTION_BLOCK T_PLC_MS_block
	VAR_OUTPUT
		T_PLC_MS :	UDINT;
	END_VAR

	VAR_EXTERNAL
		PLC_TICKS_PER_SEC :	INT;
		PLC_SYS_TICK_CNT :	DINT;
	END_VAR

	VAR
		debug :	BOOL;(*Debug-Mode ON / OFF*)
		N :	INT;(*Debug-Faktor*)
		Offset :	UDINT;(*Debug-Offset*)
		temp :	DWORD := DWORD#1;(*Debug-Offset*)
		mode :	BOOL;(*modus*)
		faktor :	UDINT;(*Systemtakt-Faktor*)
		init :	BOOL;
		v_plc_ticks_per_sec :	UDINT;
		base :	UDINT := UDINT#1000;
	END_VAR

	IF init = FALSE THEN
		v_plc_ticks_per_sec := INT_TO_UDINT(PLC_TICKS_PER_SEC);
		IF v_plc_ticks_per_sec = UDINT#1024 THEN
			faktor := UDINT#1;
			mode := FALSE;
		ELSIF v_plc_ticks_per_sec > UDINT#0 THEN
			IF v_plc_ticks_per_sec <= base THEN
				faktor := base / v_plc_ticks_per_sec;
				mode := FALSE;
			ELSE
				faktor := v_plc_ticks_per_sec / base;
				mode := TRUE;
			END_IF;
		ELSE
			faktor := UDINT#1;
		END_IF;
		init := TRUE;
	END_IF;

	IF mode THEN
		T_PLC_MS := DINT_TO_UDINT(PLC_SYS_TICK_CNT) / faktor;
	ELSE
		T_PLC_MS := DINT_TO_UDINT(PLC_SYS_TICK_CNT) * faktor;
	END_IF;

	IF debug THEN
		T_PLC_MS := (DWORD_TO_UDINT(SHL(UDINT_TO_DWORD(T_PLC_MS),N) OR SHL(temp,N)) - UDINT#1) + Offset;
	END_IF;

END_FUNCTION_BLOCK

FUNCTION TIME_TO_UDINT2:UDINT
	VAR_INPUT
		X :	TIME;
	END_VAR

	TIME_TO_UDINT2 := DINT_TO_UDINT(TIME_TO_DINT(X));
END_FUNCTION

FUNCTION FRMP_B:BYTE
	VAR_INPUT
		START :	BYTE;
		DIR :	BOOL;
		TD :	TIME;
		TR :	TIME;
	END_VAR

	IF TD < TR THEN
		FRMP_B := MIN(UDINT_TO_BYTE(DWORD_TO_UDINT(SHL(TIME_TO_DWORD(TD), 8)) / TIME_TO_UDINT2(TR)), SEL(DIR, START, USINT_TO_BYTE(USINT#255 - BYTE_TO_USINT(START))));
		IF DIR THEN
			FRMP_B := USINT_TO_BYTE(BYTE_TO_USINT(START) + BYTE_TO_USINT(FRMP_B));
		ELSE
			FRMP_B := USINT_TO_BYTE(BYTE_TO_USINT(START) - BYTE_TO_USINT(FRMP_B));
		END_IF;
	ELSE
		FRMP_B := SEL(DIR, BYTE#0, BYTE#255);
	END_IF;
END_FUNCTION

FUNCTION_BLOCK _RMP_B
	VAR_INPUT
		DIR :	BOOL;
		E :	BOOL := TRUE;
		TR :	TIME;
	END_VAR

	VAR_IN_OUT
		RMP :	BYTE;
	END_VAR

	VAR
		T_PLC_MS :	T_PLC_MS_block;
		tx :	TIME;
		tl :	TIME;
		tn :	TIME;
		init :	BOOL;
		last_dir :	BOOL;
		start :	BYTE;
	END_VAR

	T_PLC_MS();
	tx := UDINT_TO_TIME(T_PLC_MS.T_PLC_MS);

	IF E AND init AND (dir = last_dir) AND (RMP <> SEL(DIR, BYTE#0, BYTE#255)) AND TR = tn THEN
		RMP := FRMP_B(start, DIR, tx - tl, TR);
	ELSE
		init := TRUE;
		tl := tx;
		tn := tr;
		start := RMP;
	END_IF;
	last_dir := dir;
END_FUNCTION_BLOCK

FUNCTION _BYTE_TO_INT:INT
	VAR_INPUT
		IN :	BYTE;
	END_VAR

	_BYTE_TO_INT := USINT_TO_INT(BYTE_TO_USINT(IN));
END_FUNCTION

FUNCTION_BLOCK DIMM_I_Block

	VAR_INPUT
		SET :	BOOL;
		VAL :	BYTE := BYTE#255;
		IN :	BOOL;
		RST :	BOOL;
		T_DEBOUNCE :	TIME := T#10ms;
		T_RECONFIG :	TIME := T#10s;
		T_ON_MAX :	TIME := T#0h;
		T_DIMM_START :	TIME := T#1s;
		T_DIMM :	TIME := T#3s;
		MIN_ON :	BYTE := BYTE#50;
		MAX_ON :	BYTE := BYTE#255;
		SOFT_DIMM :	BOOL := TRUE;
		DBL_TOGGLE :	BOOL;
		RST_OUT :	BOOL;
	END_VAR

	VAR_OUTPUT
		Q :	BOOL;
		DBL :	BOOL;
	END_VAR

	VAR_IN_OUT
		OUT :	BYTE;
	END_VAR

	VAR
		config :	SW_RECONFIG_Block;
		decode :	CLICK_MODE_Block;
		t3 :	TON;
		dim :	_RMP_B;
		dir :	BOOL;
	END_VAR

	config(IN := IN, TD := T_DEBOUNCE, TR := T_RECONFIG);
	decode(in := config.Q, T_LONG := T_DIMM_START);

	IF RST THEN
		IF rst_out THEN out := BYTE#0; END_IF;
		Q := FALSE;
		dir := out > BYTE#127;
	ELSIF set THEN
		out := val;
		Q := TRUE;
		dir := out > BYTE#127;
	ELSIF decode.SINGLE THEN
		Q := NOT Q;
		IF Q THEN OUT := INT_TO_BYTE(LIMIT_INT(MAX(_BYTE_TO_INT(MIN_ON),1), _BYTE_TO_INT(out), _BYTE_TO_INT(MAX_ON)));	END_IF;
		dir := OUT > BYTE#127;
	ELSIF decode.TP_LONG THEN
		IF NOT Q THEN
			IF SOFT_DIMM THEN
				OUT := BYTE#1;
				dir := TRUE;
			ELSE
				out := INT_TO_BYTE(LIMIT_INT(MAX(_BYTE_TO_INT(MIN_ON),1), _BYTE_TO_INT(out), _BYTE_TO_INT(MAX_ON)));
				DIR := out < BYTE#127;
			END_IF;
			Q := TRUE;
		ELSE
			dir := NOT dir;
		END_IF;
	END_IF;

	IF NOT dbl_toggle THEN dbl := FALSE; END_IF;
	IF decode.DOUBLE THEN dbl := NOT dbl; END_IF;

	dim(DIR := dir, e := decode.LONG AND Q, TR := T_DIMM, rmp := out);
	OUT := dim.RMP;
	IF out = BYTE#0 THEN
		dir := TRUE;
	ELSIF out = BYTE#255 THEN
		dir := FALSE;
	END_IF;

	IF t_ON_MAX > t#0s THEN
		t3(in := q, pt := T_ON_MAX);
		Q := Q XOR t3.Q;
	END_IF;

END_FUNCTION_BLOCK

PROGRAM program0
	VAR
	    SET :	BOOL;
		VAL :	BYTE := BYTE#255;
		IN :	BOOL;
		RST :	BOOL;
		T_DEBOUNCE :	TIME := T#10ms;
		T_RECONFIG :	TIME := T#10s;
		T_ON_MAX :	TIME := T#0h;
		T_DIMM_START :	TIME := T#1s;
		T_DIMM :	TIME := T#3s;
		MIN_ON :	BYTE := BYTE#50;
		MAX_ON :	BYTE := BYTE#255;
		SOFT_DIMM :	BOOL := TRUE;
		DBL_TOGGLE :	BOOL;
		RST_OUT :	BOOL;
		OUT :	BYTE;
		Q :	BOOL;
		DBL :	BOOL;

		func_block : DIMM_I_Block;
  	END_VAR
	func_block.SET := SET;
	func_block.VAL := VAL;
	func_block.IN := IN;
	func_block.RST := RST;
	func_block.T_DEBOUNCE := T_DEBOUNCE;
	func_block.T_RECONFIG := T_RECONFIG;
	func_block.T_ON_MAX := T_ON_MAX;
	func_block.T_DIMM_START := T_DIMM_START;
	func_block.T_DIMM := T_DIMM;
	func_block.MIN_ON := MIN_ON;
	func_block.MAX_ON := MAX_ON;
	func_block.SOFT_DIMM := SOFT_DIMM;
	func_block.DBL_TOGGLE := DBL_TOGGLE;
	func_block.RST_OUT := RST_OUT;
	func_block.OUT := OUT;

	func_block();
	OUT := func_block.OUT;
	Q := func_block.Q;
	DBL := func_block.DBL;
END_PROGRAM

CONFIGURATION Config0
	VAR_GLOBAL
		PLC_TICKS_PER_SEC :	INT;
		PLC_SYS_TICK_CNT :	DINT;
	END_VAR
  	RESOURCE Res0 ON PLC
    	TASK task0(INTERVAL := T#20ms,PRIORITY := 0);
    	PROGRAM instance0 WITH task0 : program0;
  	END_RESOURCE
END_CONFIGURATION
